KUKA KRL program: MyProgram_250().src

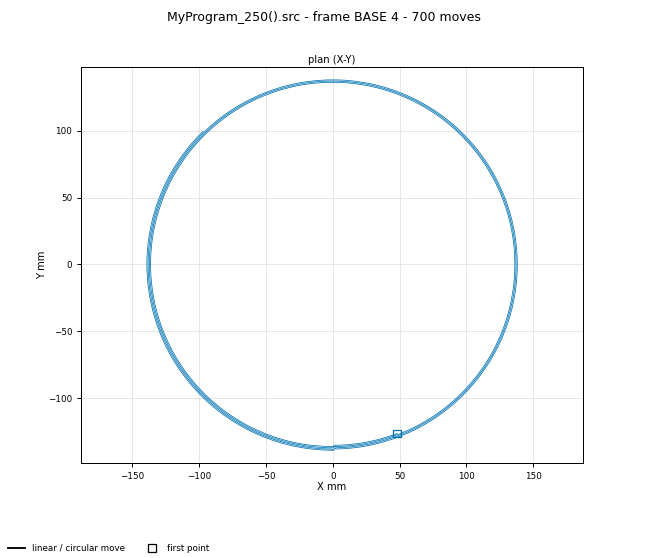
[picture p0: tool path of MyProgram_250().src in frame BASE 4, 700 of 700 moves have a stored position in this frame; points joined in program order, loops and branches not executed]
&ACCESS RVP
&REL 1
&PARAM TEMPLATE = C:\KRC\Roboter\Template\vorgabe
&PARAM EDITMASK = *
DEF MyProgram_250()
; ---- Setting reference (Base) ----
$BASE = BASE_DATA[4]

; --------------------------
; ---- Setting tool (TCP) ----
$TOOL = TOOL_DATA[3]
; --------------------------

$VEL.CP = VEL_APROX_PRINT
Startdeposition()
$VEL.CP = VEL_PRINT
LIN {X 48.2908,Y -126.5409,Z 164,A -68.332,B 12.277,C 0.2412,E1 12.3361,E2 518.7621} C_DIS
LIN {X 45.6625,Y -127.5105,Z 164,A -69.5545,B 12.2769,C 0.2436,E1 12.3329,E2 519.99} C_DIS
LIN {X 42.0708,Y -128.7422,Z 164,A -71.1085,B 12.2769,C 0.2439,E1 12.3288,E2 521.5389} C_DIS
LIN {X 38.9153,Y -129.7308,Z 164,A -72.4885,B 12.2769,C 0.2447,E1 12.3251,E2 522.9177} C_DIS
LIN {X 35.7562,Y -130.6369,Z 164,A -73.8812,B 12.2769,C 0.2461,E1 12.3214,E2 524.3117} C_DIS
LIN {X 32.9488,Y -131.3715,Z 164,A -75.1311,B 12.2769,C 0.2478,E1 12.318,E2 525.5653} C_DIS
LIN {X 29.371,Y -132.2193,Z 164,A -76.6506,B 12.2768,C 0.248,E1 12.3139,E2 527.0815} C_DIS
LIN {X 26.2188,Y -132.8803,Z 164,A -78.0066,B 12.2768,C 0.2489,E1 12.3102,E2 528.4377} C_DIS
LIN {X 23.2474,Y -133.4313,Z 164,A -79.2594,B 12.2768,C 0.249,E1 12.3067,E2 529.688} C_DIS
LIN {X 19.9409,Y -133.9663,Z 164,A -80.6907,B 12.2768,C 0.2502,E1 12.3028,E2 531.1221} C_DIS
LIN {X 16.8205,Y -134.3937,Z 164,A -82.0176,B 12.2768,C 0.2508,E1 12.2991,E2 532.4492} C_DIS
LIN {X 13.7158,Y -134.746,Z 164,A -83.3348,B 12.2768,C 0.2513,E1 12.2954,E2 533.7665} C_DIS
LIN {X 10.87,Y -135.0042,Z 164,A -84.525,B 12.2768,C 0.2513,E1 12.2921,E2 534.9551} C_DIS
LIN {X 7.9689,Y -135.2059,Z 164,A -85.7974,B 12.2768,C 0.2528,E1 12.2886,E2 536.2334} C_DIS
LIN {X 4.5191,Y -135.3668,Z 164,A -87.2223,B 12.2768,C 0.2522,E1 12.2846,E2 537.6546} C_DIS
LIN {X 0.9829,Y -135.4364,Z 164,A -88.496,B 12.2768,C 0.2465,E1 12.2811,E2 538.9014} C_DIS
Enddeposition()
LIN {X 0.9829,Y -135.4364,Z 164,A -88.496,B 12.2768,C 0.2465,E1 12.2811,E2 538.9014} C_DIS
Startdeposition()
$VEL.CP = VEL_PRINT
LIN {X 1.1754,Y -136.3554,Z 164,A -87.5778,B 12.2004,C 0.236,E1 12.2073,E2 537.9358} C_DIS
LIN {X 5.011,Y -136.268,Z 164,A -86.5742,B 12.2001,C 0.252,E1 12.2098,E2 537.0086} C_DIS
LIN {X 9.3611,Y -136.0392,Z 164,A -84.1098,B 12.2004,C 0.2343,E1 12.2169,E2 534.4629} C_DIS
LIN {X 13.3056,Y -135.7092,Z 164,A -82.8957,B 12.2002,C 0.2458,E1 12.2201,E2 533.3049} C_DIS
LIN {X 17.0554,Y -135.2905,Z 164,A -81.1665,B 12.2002,C 0.2411,E1 12.2249,E2 531.5566} C_DIS
LIN {X 20.8387,Y -134.7579,Z 164,A -79.6734,B 12.2002,C 0.2433,E1 12.229,E2 530.0767} C_DIS
LIN {X 24.8084,Y -134.0861,Z 164,A -77.9252,B 12.2003,C 0.2406,E1 12.2338,E2 528.3202} C_DIS
LIN {X 27.9166,Y -133.4733,Z 164,A -76.7034,B 12.2003,C 0.2427,E1 12.2372,E2 527.1114} C_DIS
LIN {X 30.4077,Y -132.9258,Z 164,A -75.5929,B 12.2003,C 0.2407,E1 12.2402,E2 525.9951} C_DIS
LIN {X 33.7097,Y -132.1272,Z 164,A -74.1914,B 12.2003,C 0.2402,E1 12.244,E2 524.5958} C_DIS
LIN {X 36.6449,Y -131.3432,Z 164,A -72.8971,B 12.2003,C 0.2386,E1 12.2475,E2 523.2983} C_DIS
LIN {X 40.6848,Y -130.1509,Z 164,A -71.1725,B 12.2003,C 0.2381,E1 12.2521,E2 521.5782} C_DIS
LIN {X 43.4948,Y -129.2373,Z 164,A -69.9381,B 12.2003,C 0.237,E1 12.2554,E2 520.3436} C_DIS
LIN {X 46.722,Y -128.1061,Z 164,A -68.506,B 12.2004,C 0.2355,E1 12.2591,E2 518.9109} C_DIS
LIN {X 49.6795,Y -126.9878,Z 164,A -67.1784,B 12.2004,C 0.2339,E1 12.2626,E2 517.5824} C_DIS
LIN {X 53.377,Y -125.4806,Z 164,A -65.5189,B 12.2004,C 0.2323,E1 12.2669,E2 515.9237} C_DIS
LIN {X 56.1528,Y -124.2617,Z 164,A -64.2407,B 12.2005,C 0.2305,E1 12.2701,E2 514.6438} C_DIS
LIN {X 60.2052,Y -122.3486,Z 164,A -62.1678,B 12.2006,C 0.2225,E1 12.2754,E2 512.5451} C_DIS
LIN {X 64.1876,Y -120.31,Z 164,A -60.4796,B 12.2006,C 0.2251,E1 12.2795,E2 510.8796} C_DIS
LIN {X 67.2225,Y -118.6409,Z 164,A -58.9313,B 12.2006,C 0.2202,E1 12.2833,E2 509.318} C_DIS
LIN {X 71.1825,Y -116.3076,Z 164,A -57.0303,B 12.2007,C 0.2179,E1 12.2879,E2 507.419} C_DIS
LIN {X 76.8995,Y -112.6097,Z 164,A -54.2881,B 12.2007,C 0.2164,E1 12.2943,E2 504.689} C_DIS
LIN {X 80.1373,Y -110.3286,Z 164,A -52.5882,B 12.2008,C 0.2123,E1 12.2981,E2 502.9829} C_DIS
LIN {X 83.4574,Y -107.839,Z 164,A -50.8412,B 12.2008,C 0.2089,E1 12.302,E2 501.2336} C_DIS
LIN {X 86.7001,Y -105.2501,Z 164,A -49.0457,B 12.201,C 0.2039,E1 12.3059,E2 499.4297} C_DIS
LIN {X 90.2463,Y -102.2252,Z 164,A -47.1321,B 12.201,C 0.2012,E1 12.3099,E2 497.5197} C_DIS
LIN {X 93.5477,Y -99.2129,Z 164,A -45.3151,B 12.201,C 0.199,E1 12.3136,E2 495.7083} C_DIS
LIN {X 96.533,Y -96.3111,Z 164,A -43.5592,B 12.2011,C 0.1951,E1 12.3171,E2 493.9497} C_DIS
LIN {X 99.5558,Y -93.1834,Z 164,A -41.2789,B 12.2014,C 0.1777,E1 12.3216,E2 491.6097} C_DIS
LIN {X 102.6887,Y -89.7185,Z 164,A -39.8828,B 12.2012,C 0.1898,E1 12.3241,E2 490.2835} C_DIS
LIN {X 106.8768,Y -84.6866,Z 164,A -37.2703,B 12.2012,C 0.1873,E1 12.3287,E2 487.6854} C_DIS
LIN {X 110.0508,Y -80.5187,Z 164,A -34.9862,B 12.2013,C 0.1796,E1 12.3326,E2 485.3884} C_DIS
LIN {X 112.1141,Y -77.6202,Z 164,A -33.4583,B 12.2014,C 0.1749,E1 12.335,E2 483.8546} C_DIS
LIN {X 114.4786,Y -74.0883,Z 164,A -31.6477,B 12.2014,C 0.1696,E1 12.3378,E2 482.0387} C_DIS
LIN {X 116.7798,Y -70.4053,Z 164,A -29.8574,B 12.2015,C 0.1659,E1 12.3404,E2 480.2506} C_DIS
LIN {X 118.8236,Y -66.898,Z 164,A -28.1541,B 12.2015,C 0.1615,E1 12.3428,E2 478.5456} C_DIS
LIN {X 121.0055,Y -62.8639,Z 164,A -26.1017,B 12.2017,C 0.1526,E1 12.3455,E2 476.4749} C_DIS
LIN {X 123.7331,Y -57.3059,Z 164,A -23.6996,B 12.2017,C 0.1514,E1 12.3483,E2 474.0949} C_DIS
LIN {X 125.3016,Y -53.7911,Z 164,A -22.153,B 12.2017,C 0.149,E1 12.3501,E2 472.5554} C_DIS
LIN {X 126.9426,Y -49.7956,Z 164,A -20.1796,B 12.2019,C 0.1393,E1 12.3521,E2 470.5597} C_DIS
LIN {X 128.4672,Y -45.7204,Z 164,A -18.565,B 12.2019,C 0.1405,E1 12.3536,E2 468.9701} C_DIS
LIN {X 129.6221,Y -42.339,Z 164,A -16.9303,B 12.2019,C 0.1322,E1 12.3551,E2 467.3168} C_DIS
LIN {X 130.8644,Y -38.3198,Z 164,A -15.3357,B 12.2019,C 0.1322,E1 12.3564,E2 465.7418} C_DIS
LIN {X 131.7544,Y -35.138,Z 164,A -13.9371,B 12.2019,C 0.128,E1 12.3574,E2 464.3403} C_DIS
LIN {X 132.7794,Y -31.0487,Z 164,A -12.2707,B 12.202,C 0.1259,E1 12.3585,E2 462.6851} C_DIS
LIN {X 133.6162,Y -27.2146,Z 164,A -10.3755,B 12.2021,C 0.1138,E1 12.3596,E2 460.7568} C_DIS
LIN {X 134.5659,Y -22.0482,Z 164,A -8.5679,B 12.2021,C 0.1192,E1 12.3605,E2 458.9971} C_DIS
LIN {X 134.9692,Y -19.4238,Z 164,A -7.2771,B 12.2021,C 0.1107,E1 12.361,E2 457.6829} C_DIS
LIN {X 135.4378,Y -15.8324,Z 164,A -5.6973,B 12.2022,C 0.1045,E1 12.3615,E2 456.0941} C_DIS
LIN {X 135.9509,Y -10.5712,Z 164,A -3.3772,B 12.2022,C 0.095,E1 12.3621,E2 453.7591} C_DIS
LIN {X 136.2584,Y -5.2565,Z 164,A -1.3986,B 12.2022,C 0.096,E1 12.3624,E2 451.8104} C_DIS
LIN {X 136.3511,Y -1.6569,Z 164,A 0.6013,B 12.2024,C 0.077,E1 12.3624,E2 449.7474} C_DIS
LIN {X 136.3329,Y 2.7517,Z 164,A 2.035,B 12.2024,C 0.084,E1 12.3624,E2 448.3646} C_DIS
LIN {X 136.0966,Y 8.4677,Z 164,A 4.3122,B 12.2024,C 0.0807,E1 12.3621,E2 446.1008} C_DIS
LIN {X 135.8407,Y 11.8936,Z 164,A 5.7832,B 12.2024,C 0.0756,E1 12.3617,E2 444.6249} C_DIS
LIN {X 135.3747,Y 16.3615,Z 164,A 7.552,B 12.2024,C 0.0736,E1 12.3612,E2 442.8689} C_DIS
LIN {X 134.8736,Y 20.0915,Z 164,A 9.3282,B 12.2024,C 0.0632,E1 12.3605,E2 441.0667} C_DIS
LIN {X 134.2268,Y 24.023,Z 164,A 10.8118,B 12.2024,C 0.064,E1 12.3598,E2 439.6054} C_DIS
LIN {X 133.6003,Y 27.2926,Z 164,A 12.2295,B 12.2025,C 0.0594,E1 12.359,E2 438.1839} C_DIS
LIN {X 132.8339,Y 30.8104,Z 164,A 13.82,B 12.2025,C 0.0528,E1 12.358,E2 436.5822} C_DIS
LIN {X 131.7281,Y 35.2364,Z 164,A 15.6314,B 12.2025,C 0.0504,E1 12.3568,E2 434.7822} C_DIS
LIN {X 130.7907,Y 38.5714,Z 164,A 17.007,B 12.2025,C 0.0487,E1 12.3557,E2 433.4153} C_DIS
LIN {X 129.6256,Y 42.3281,Z 164,A 18.626,B 12.2025,C 0.045,E1 12.3543,E2 431.7991} C_DIS
LIN {X 128.6051,Y 45.3331,Z 164,A 20.2475,B 12.2026,C 0.0329,E1 12.3528,E2 430.1404} C_DIS
LIN {X 126.6777,Y 50.467,Z 164,A 22.1375,B 12.2026,C 0.0387,E1 12.351,E2 428.3001} C_DIS
LIN {X 125.2088,Y 54.0057,Z 164,A 23.8065,B 12.2026,C 0.0326,E1 12.3492,E2 426.6224} C_DIS
LIN {X 123.8611,Y 57.029,Z 164,A 25.2775,B 12.2026,C 0.0266,E1 12.3474,E2 425.1403} C_DIS
LIN {X 122.1015,Y 60.7062,Z 164,A 26.9507,B 12.2026,C 0.0233,E1 12.3454,E2 423.4708} C_DIS
LIN {X 119.9975,Y 64.7693,Z 164,A 29.0703,B 12.2026,C 0.0126,E1 12.3426,E2 421.3252} C_DIS
LIN {X 117.4266,Y 69.3215,Z 164,A 31.0431,B 12.2026,C 0.0136,E1 12.3399,E2 419.3788} C_DIS
LIN {X 115.3058,Y 72.7938,Z 164,A 32.7303,B 12.2026,C 0.01,E1 12.3374,E2 417.6932} C_DIS
LIN {X 113.0619,Y 76.2328,Z 164,A 34.4602,B 12.2026,C 0.0057,E1 12.3347,E2 415.9616} C_DIS
LIN {X 110.1487,Y 80.3855,Z 164,A 36.5792,B 12.2026,C 0.001,E1 12.3313,E2 413.843} C_DIS
LIN {X 107.5201,Y 83.8688,Z 164,A 38.3945,B 12.2026,C -0.0027,E1 12.3282,E2 412.0288} C_DIS
LIN {X 104.8808,Y 87.1461,Z 164,A 40.1189,B 12.2026,C -0.0054,E1 12.3251,E2 410.3089} C_DIS
LIN {X 102.0458,Y 90.4492,Z 164,A 42.1318,B 12.2026,C -0.0147,E1 12.3214,E2 408.2722} C_DIS
LIN {X 99.2051,Y 93.556,Z 164,A 43.6393,B 12.2026,C -0.011,E1 12.3186,E2 406.7963} C_DIS
LIN {X 96.6273,Y 96.2162,Z 164,A 45.2671,B 12.2026,C -0.0162,E1 12.3154,E2 405.159} C_DIS
LIN {X 93.3106,Y 99.4366,Z 164,A 47.1839,B 12.2026,C -0.0193,E1 12.3115,E2 403.2445} C_DIS
LIN {X 90.041,Y 102.4067,Z 164,A 49.0558,B 12.2026,C -0.0233,E1 12.3076,E2 401.3699} C_DIS
LIN {X 82.6384,Y 108.4682,Z 164,A 52.8958,B 12.2026,C -0.0254,E1 12.2993,E2 397.5512} C_DIS
LIN {X 79.2735,Y 110.9509,Z 164,A 54.7025,B 12.2026,C -0.0298,E1 12.2952,E2 395.738} C_DIS
LIN {X 76.0068,Y 113.2143,Z 164,A 56.4444,B 12.2026,C -0.0345,E1 12.2912,E2 393.9867} C_DIS
LIN {X 72.4317,Y 115.5344,Z 164,A 58.2319,B 12.2026,C -0.0371,E1 12.287,E2 392.1994} C_DIS
LIN {X 68.7576,Y 117.7578,Z 164,A 60.021,B 12.2026,C -0.0393,E1 12.2827,E2 390.4118} C_DIS
LIN {X 64.8699,Y 119.9434,Z 164,A 61.8995,B 12.2026,C -0.042,E1 12.2781,E2 388.5325} C_DIS
LIN {X 60.8693,Y 122.021,Z 164,A 63.5625,B 12.2026,C -0.0381,E1 12.274,E2 386.8979} C_DIS
LIN {X 58.5741,Y 123.138,Z 164,A 64.7213,B 12.2026,C -0.0418,E1 12.2711,E2 385.7283} C_DIS
LIN {X 55.6269,Y 124.497,Z 164,A 66.0594,B 12.2026,C -0.0427,E1 12.2677,E2 384.3934} C_DIS
LIN {X 48.0521,Y 127.6123,Z 164,A 69.4891,B 12.2026,C -0.0459,E1 12.2588,E2 380.9654} C_DIS
LIN {X 43.7055,Y 129.1671,Z 164,A 71.365,B 12.2026,C -0.0459,E1 12.2539,E2 379.0976} C_DIS
LIN {X 40.232,Y 130.2896,Z 164,A 73.0275,B 12.2026,C -0.0507,E1 12.2494,E2 377.4195} C_DIS
LIN {X 36.7393,Y 131.3168,Z 164,A 74.5177,B 12.2026,C -0.0508,E1 12.2454,E2 375.9343} C_DIS
LIN {X 33.2881,Y 132.2341,Z 164,A 75.9811,B 12.2026,C -0.0508,E1 12.2415,E2 374.4757} C_DIS
LIN {X 29.6047,Y 133.1093,Z 164,A 77.5547,B 12.2026,C -0.0513,E1 12.2372,E2 372.9046} C_DIS
LIN {X 26.7382,Y 133.7131,Z 164,A 78.9283,B 12.2026,C -0.0558,E1 12.2334,E2 371.5138} C_DIS
LIN {X 20.8769,Y 134.752,Z 164,A 81.361,B 12.2026,C -0.055,E1 12.2267,E2 369.0902} C_DIS
LIN {X 17.6083,Y 135.218,Z 164,A 82.6906,B 12.2026,C -0.054,E1 12.2231,E2 367.7681} C_DIS
LIN {X 14.3853,Y 135.5989,Z 164,A 84.1121,B 12.2026,C -0.0559,E1 12.2191,E2 366.3399} C_DIS
LIN {X 9.93,Y 135.9977,Z 164,A 86.277,B 12.2025,C -0.0637,E1 12.213,E2 364.1407} C_DIS
LIN {X 6.2453,Y 136.218,Z 164,A 87.5863,B 12.2025,C -0.0575,E1 12.2094,E2 362.8618} C_DIS
LIN {X 2.09,Y 136.3439,Z 164,A 89.2131,B 12.2025,C -0.0544,E1 12.2049,E2 361.2504} C_DIS
LIN {X -2.8802,Y 136.3305,Z 164,A 91.4358,B 12.2025,C -0.0576,E1 12.1987,E2 359.0123} C_DIS
LIN {X -6.0127,Y 136.2289,Z 164,A 92.6748,B 12.2025,C -0.0554,E1 12.1952,E2 357.7837} C_DIS
LIN {X -9.8724,Y 136.0019,Z 164,A 94.2822,B 12.2025,C -0.0545,E1 12.1908,E2 356.1791} C_DIS
LIN {X -13.5412,Y 135.6866,Z 164,A 96.1288,B 12.2025,C -0.0617,E1 12.1855,E2 354.2968} C_DIS
LIN {X -17.0169,Y 135.2955,Z 164,A 97.2229,B 12.2025,C -0.0514,E1 12.1826,E2 353.2496} C_DIS
LIN {X -21.6342,Y 134.6347,Z 164,A 99.2182,B 12.2025,C -0.0514,E1 12.1771,E2 351.2512} C_DIS
LIN {X -25.9034,Y 133.8769,Z 164,A 101.1442,B 12.2025,C -0.0529,E1 12.1718,E2 349.3135} C_DIS
LIN {X -29.3192,Y 133.1713,Z 164,A 102.4765,B 12.2025,C -0.0485,E1 12.1682,E2 347.9986} C_DIS
LIN {X -31.9571,Y 132.5619,Z 164,A 103.6842,B 12.2025,C -0.0495,E1 12.1649,E2 346.7831} C_DIS
LIN {X -35.489,Y 131.6608,Z 164,A 105.1942,B 12.2025,C -0.0477,E1 12.1608,E2 345.2769} C_DIS
LIN {X -38.2408,Y 130.8875,Z 164,A 106.4065,B 12.2025,C -0.0469,E1 12.1576,E2 344.0641} C_DIS
LIN {X -41.5848,Y 129.8637,Z 164,A 108.3021,B 12.2025,C -0.0562,E1 12.1524,E2 342.1174} C_DIS
LIN {X -45.3778,Y 128.5896,Z 164,A 109.5797,B 12.2025,C -0.0443,E1 12.1491,E2 340.8907} C_DIS
LIN {X -48.6915,Y 127.3718,Z 164,A 111.2139,B 12.2025,C -0.0464,E1 12.1448,E2 339.2392} C_DIS
LIN {X -53.357,Y 125.4893,Z 164,A 113.1901,B 12.2025,C -0.0405,E1 12.1398,E2 337.2817} C_DIS
LIN {X -57.4791,Y 123.653,Z 164,A 115.1186,B 12.2025,C -0.0389,E1 12.1349,E2 335.3508} C_DIS
LIN {X -60.6509,Y 122.1288,Z 164,A 116.6044,B 12.2025,C -0.0371,E1 12.1311,E2 333.8655} C_DIS
LIN {X -64.1634,Y 120.3223,Z 164,A 118.1754,B 12.2026,C -0.0325,E1 12.1273,E2 332.3068} C_DIS
LIN {X -67.1054,Y 118.707,Z 164,A 119.7535,B 12.2026,C -0.0345,E1 12.1234,E2 330.7097} C_DIS
LIN {X -70.5956,Y 116.6647,Z 164,A 121.5191,B 12.2026,C -0.0335,E1 12.1191,E2 328.9376} C_DIS
LIN {X -75.2515,Y 113.7176,Z 164,A 123.5708,B 12.2026,C -0.0232,E1 12.1144,E2 326.9203} C_DIS
LIN {X -77.6775,Y 112.0743,Z 164,A 125.0837,B 12.2026,C -0.0279,E1 12.1108,E2 325.3742} C_DIS
LIN {X -81.3795,Y 109.4156,Z 164,A 127.1729,B 12.2026,C -0.0286,E1 12.1061,E2 323.2657} C_DIS
LIN {X -86.4616,Y 105.4458,Z 164,A 129.6546,B 12.2026,C -0.018,E1 12.1007,E2 320.8148} C_DIS
LIN {X -89.6471,Y 102.751,Z 164,A 131.4544,B 12.2026,C -0.0157,E1 12.0969,E2 319.0112} C_DIS
LIN {X -93.98,Y 98.804,Z 164,A 134.1578,B 12.2026,C -0.0163,E1 12.0913,E2 316.281} C_DIS
LIN {X -97.8786,Y 94.943,Z 164,A 136.2674,B 12.2026,C -0.0067,E1 12.0872,E2 314.1978} C_DIS
LIN {X -100.6527,Y 91.9976,Z 164,A 138.1624,B 12.2026,C -0.0075,E1 12.0836,E2 312.2809} C_DIS
LIN {X -103.5079,Y 88.7726,Z 164,A 139.7765,B 12.2026,C 0.0012,E1 12.0807,E2 310.6929} C_DIS
LIN {X -105.9909,Y 85.7926,Z 164,A 141.464,B 12.2026,C 0.0037,E1 12.0777,E2 309.0001} C_DIS
LIN {X -108.3883,Y 82.7427,Z 164,A 143.1293,B 12.2026,C 0.0067,E1 12.0748,E2 307.3324} C_DIS
LIN {X -110.9239,Y 79.3113,Z 164,A 144.9088,B 12.2026,C 0.0114,E1 12.0719,E2 305.5566} C_DIS
LIN {X -113.3119,Y 75.8606,Z 164,A 146.7387,B 12.2026,C 0.0143,E1 12.069,E2 303.7206} C_DIS
LIN {X -115.7364,Y 72.1074,Z 164,A 148.596,B 12.2026,C 0.0195,E1 12.0663,E2 301.868} C_DIS
LIN {X -117.8522,Y 68.5955,Z 164,A 150.3387,B 12.2026,C 0.0235,E1 12.0638,E2 300.1248} C_DIS
LIN {X -119.9202,Y 64.9131,Z 164,A 152.1972,B 12.2026,C 0.0262,E1 12.0613,E2 298.2582} C_DIS
LIN {X -121.7494,Y 61.4099,Z 164,A 153.7585,B 12.2026,C 0.0329,E1 12.0593,E2 296.711} C_DIS
LIN {X -123.1428,Y 58.5641,Z 164,A 155.0945,B 12.2026,C 0.0364,E1 12.0577,E2 295.376} C_DIS
LIN {X -124.7097,Y 55.1514,Z 164,A 156.6981,B 12.2026,C 0.0401,E1 12.0559,E2 293.7711} C_DIS
LIN {X -125.9443,Y 52.2683,Z 164,A 157.9973,B 12.2026,C 0.0442,E1 12.0544,E2 292.4757} C_DIS
LIN {X -127.3,Y 48.8763,Z 164,A 159.7004,B 12.2026,C 0.0446,E1 12.0527,E2 290.7538} C_DIS
LIN {X -130.2844,Y 40.2492,Z 164,A 163.2741,B 12.2025,C 0.0615,E1 12.0495,E2 287.217} C_DIS
LIN {X -131.6813,Y 35.4122,Z 164,A 165.3884,B 12.2025,C 0.0676,E1 12.0479,E2 285.1055} C_DIS
LIN {X -132.2734,Y 33.1333,Z 164,A 166.5437,B 12.2025,C 0.0667,E1 12.0471,E2 283.931} C_DIS
LIN {X -133.0087,Y 30.0448,Z 164,A 167.9427,B 12.2025,C 0.0691,E1 12.0462,E2 282.5256} C_DIS
LIN {X -133.7746,Y 26.4358,Z 164,A 169.6736,B 12.2025,C 0.0694,E1 12.0452,E2 280.7743} C_DIS
LIN {X -134.4969,Y 22.4613,Z 164,A 171.2578,B 12.2025,C 0.077,E1 12.0445,E2 279.2059} C_DIS
LIN {X -135.1097,Y 18.4347,Z 164,A 172.9444,B 12.2024,C 0.0826,E1 12.0438,E2 277.5244} C_DIS
LIN {X -135.5574,Y 14.7708,Z 164,A 174.654,B 12.2024,C 0.0835,E1 12.0433,E2 275.797} C_DIS
LIN {X -135.8857,Y 11.3605,Z 164,A 176.0931,B 12.2024,C 0.0878,E1 12.0429,E2 274.3596} C_DIS
LIN {X -136.1893,Y 6.8168,Z 164,A 177.9499,B 12.2023,C 0.0948,E1 12.0426,E2 272.5119} C_DIS
LIN {X -136.3248,Y 3.1531,Z 164,A 179.4669,B 12.2023,C 0.0999,E1 12.0425,E2 270.9995} C_DIS
LIN {X -136.3582,Y -0.6868,Z 164,A -178.8085,B 12.2023,C 0.1021,E1 12.0425,E2 269.2629} C_DIS
LIN {X -136.2686,Y -4.9965,Z 164,A -176.9851,B 12.2022,C 0.1072,E1 12.0426,E2 267.44} C_DIS
LIN {X -136.0777,Y -8.7749,Z 164,A -175.4217,B 12.2022,C 0.1124,E1 12.0429,E2 265.8816} C_DIS
LIN {X -135.7422,Y -12.9626,Z 164,A -173.6138,B 12.2021,C 0.1167,E1 12.0433,E2 264.0702} C_DIS
LIN {X -135.3736,Y -16.3707,Z 164,A -172.2277,B 12.2021,C 0.1221,E1 12.0437,E2 262.6923} C_DIS
LIN {X -134.944,Y -19.6,Z 164,A -170.768,B 12.2021,C 0.124,E1 12.0443,E2 261.2228} C_DIS
LIN {X -134.4164,Y -22.9437,Z 164,A -169.3405,B 12.202,C 0.128,E1 12.0449,E2 259.7961} C_DIS
LIN {X -133.6599,Y -26.9997,Z 164,A -167.5657,B 12.202,C 0.1321,E1 12.0459,E2 258.0179} C_DIS
LIN {X -132.8522,Y -30.73,Z 164,A -165.9037,B 12.202,C 0.1353,E1 12.0469,E2 256.3502} C_DIS
LIN {X -130.8835,Y -38.2546,Z 164,A -162.7074,B 12.2018,C 0.1463,E1 12.0492,E2 253.166} C_DIS
LIN {X -129.7971,Y -41.7935,Z 164,A -161.0607,B 12.2018,C 0.1485,E1 12.0506,E2 251.5094} C_DIS
LIN {X -128.1723,Y -46.5385,Z 164,A -158.8901,B 12.2018,C 0.1528,E1 12.0526,E2 249.3328} C_DIS
LIN {X -126.8925,Y -49.9245,Z 164,A -157.42,B 12.2016,C 0.1581,E1 12.0541,E2 247.8704} C_DIS
LIN {X -125.6054,Y -53.0798,Z 164,A -155.965,B 12.2016,C 0.1614,E1 12.0556,E2 246.4137} C_DIS
LIN {X -124.319,Y -56.0248,Z 164,A -154.1259,B 12.2016,C 0.1535,E1 12.0578,E2 244.5146} C_DIS
LIN {X -122.5111,Y -59.8758,Z 164,A -152.9286,B 12.2015,C 0.1721,E1 12.0592,E2 243.3924} C_DIS
LIN {X -121.5055,Y -61.8889,Z 164,A -151.8691,B 12.2015,C 0.1719,E1 12.0605,E2 242.3194} C_DIS
LIN {X -119.8259,Y -65.0861,Z 164,A -150.3428,B 12.2015,C 0.1756,E1 12.0625,E2 240.7932} C_DIS
LIN {X -117.9612,Y -68.4073,Z 164,A -148.5971,B 12.2014,C 0.1761,E1 12.065,E2 239.0307} C_DIS
LIN {X -115.6313,Y -72.2763,Z 164,A -146.666,B 12.2014,C 0.18,E1 12.0678,E2 237.0966} C_DIS
LIN {X -112.3824,Y -77.2308,Z 164,A -144.1988,B 12.2012,C 0.1865,E1 12.0716,E2 234.6339} C_DIS
LIN {X -109.8492,Y -80.7932,Z 164,A -142.2985,B 12.2012,C 0.1893,E1 12.0747,E2 232.7267} C_DIS
LIN {X -107.3054,Y -84.1424,Z 164,A -140.5351,B 12.2012,C 0.1934,E1 12.0778,E2 230.9649} C_DIS
LIN {X -104.5833,Y -87.5028,Z 164,A -138.593,B 12.2012,C 0.1944,E1 12.0812,E2 229.0081} C_DIS
LIN {X -102.3766,Y -90.075,Z 164,A -137.2836,B 12.201,C 0.2002,E1 12.0836,E2 227.7139} C_DIS
LIN {X -99.6679,Y -93.063,Z 164,A -135.57,B 12.201,C 0.2033,E1 12.0869,E2 225.9987} C_DIS
LIN {X -97.0183,Y -95.8227,Z 164,A -133.8879,B 12.201,C 0.2047,E1 12.0902,E2 224.3079} C_DIS
LIN {X -94.0628,Y -98.7249,Z 164,A -132.156,B 12.2009,C 0.2084,E1 12.0936,E2 222.5778} C_DIS
LIN {X -90.772,Y -101.759,Z 164,A -129.7114,B 12.2011,C 0.198,E1 12.0989,E2 220.0629} C_DIS
LIN {X -86.8596,Y -105.1181,Z 164,A -128.5277,B 12.2006,C 0.2261,E1 12.1011,E2 219.0035} C_DIS
LIN {X -83.2535,Y -107.997,Z 164,A -126.071,B 12.2007,C 0.2168,E1 12.1067,E2 216.4827} C_DIS
LIN {X -79.5121,Y -110.7802,Z 164,A -124.1355,B 12.2007,C 0.2206,E1 12.111,E2 214.5507} C_DIS
LIN {X -75.7632,Y -113.3769,Z 164,A -122.2299,B 12.2007,C 0.2238,E1 12.1154,E2 212.6468} C_DIS
LIN {X -72.1239,Y -115.7261,Z 164,A -120.4363,B 12.2006,C 0.2272,E1 12.1196,E2 210.8569} C_DIS
LIN {X -68.6534,Y -117.8187,Z 164,A -118.6976,B 12.2006,C 0.2287,E1 12.1238,E2 209.1139} C_DIS
LIN {X -64.8019,Y -119.9799,Z 164,A -116.7819,B 12.2006,C 0.2296,E1 12.1285,E2 207.1908} C_DIS
LIN {X -61.5596,Y -121.6732,Z 164,A -115.3776,B 12.2004,C 0.2348,E1 12.132,E2 205.8033} C_DIS
LIN {X -58.4721,Y -123.1867,Z 164,A -113.9328,B 12.2004,C 0.2365,E1 12.1356,E2 204.3586} C_DIS
LIN {X -50.3113,Y -126.7405,Z 164,A -110.2336,B 12.2003,C 0.2415,E1 12.1451,E2 200.6648} C_DIS
LIN {X -46.8174,Y -128.0717,Z 164,A -108.6754,B 12.2003,C 0.2433,E1 12.1492,E2 199.1082} C_DIS
LIN {X -43.4067,Y -129.2666,Z 164,A -106.9843,B 12.2003,C 0.2401,E1 12.1537,E2 197.3951} C_DIS
LIN {X -39.9183,Y -130.3856,Z 164,A -105.4121,B 12.2003,C 0.2404,E1 12.1579,E2 195.8186} C_DIS
LIN {X -34.7412,Y -131.8602,Z 164,A -103.248,B 12.2003,C 0.2444,E1 12.1637,E2 193.6665} C_DIS
LIN {X -31.5292,Y -132.665,Z 164,A -101.7848,B 12.2003,C 0.2433,E1 12.1677,E2 192.1939} C_DIS
LIN {X -27.3737,Y -133.5838,Z 164,A -99.6321,B 12.2004,C 0.2346,E1 12.1737,E2 189.9945} C_DIS
LIN {X -23.3491,Y -134.3473,Z 164,A -98.3049,B 12.2002,C 0.2457,E1 12.1772,E2 188.7169} C_DIS
LIN {X -19.2093,Y -134.9998,Z 164,A -96.5759,B 12.2002,C 0.247,E1 12.182,E2 186.9914} C_DIS
LIN {X -15.5778,Y -135.4681,Z 164,A -94.7869,B 12.2003,C 0.2408,E1 12.187,E2 185.1701} C_DIS
LIN {X -5.7775,Y -136.2381,Z 164,A -91.0439,B 12.2001,C 0.2514,E1 12.1973,E2 181.4747} C_DIS
LIN {X 0.9712,Y -136.3528,Z 164,A -89.3946,B 12.1994,C 0.2826,E1 12.2016,E2 179.9726} C_DIS
Enddeposition()
LIN {X 0.9712,Y -136.3528,Z 164,A -89.3948,B 12.1994,C 0.2826,E1 12.2016,E2 179.9728} C_DIS
Startdeposition()
$VEL.CP = VEL_PRINT
LIN {X 0.6652,Y -137.2779,Z 164,A -89.4096,B 12.1186,C 0.2916,E1 12.1208,E2 180.0344} C_DIS
LIN {X -4.5946,Y -137.2046,Z 164,A -91.0487,B 12.119,C 0.2772,E1 12.1164,E2 181.6049} C_DIS
LIN {X -7.9431,Y -137.0503,Z 164,A -92.7499,B 12.1188,C 0.285,E1 12.1115,E2 183.3447} C_DIS
LIN {X -11.6534,Y -136.7839,Z 164,A -93.9544,B 12.119,C 0.2758,E1 12.1083,E2 184.5061} C_DIS
LIN {X -17.3961,Y -136.1733,Z 164,A -96.3368,B 12.119,C 0.2746,E1 12.1017,E2 186.8858} C_DIS
LIN {X -20.6764,Y -135.7136,Z 164,A -98.8778,B 12.1183,C 0.304,E1 12.0943,E2 189.5716} C_DIS
LIN {X -28.5232,Y -134.284,Z 164,A -101.1177,B 12.119,C 0.2746,E1 12.0885,E2 191.6769} C_DIS
LIN {X -32.0412,Y -133.4876,Z 164,A -102.5474,B 12.119,C 0.2719,E1 12.0846,E2 193.0975} C_DIS
LIN {X -35.6795,Y -132.5618,Z 164,A -104.1585,B 12.119,C 0.272,E1 12.0803,E2 194.7145} C_DIS
LIN {X -39.8501,Y -131.3682,Z 164,A -105.965,B 12.1191,C 0.2707,E1 12.0754,E2 196.5207} C_DIS
LIN {X -43.2788,Y -130.2785,Z 164,A -107.4134,B 12.1191,C 0.2681,E1 12.0716,E2 197.9625} C_DIS
LIN {X -45.9692,Y -129.3551,Z 164,A -108.6792,B 12.1191,C 0.2691,E1 12.0682,E2 199.2385} C_DIS
LIN {X -49.2116,Y -128.1563,Z 164,A -110.1493,B 12.1191,C 0.2685,E1 12.0644,E2 200.712} C_DIS
LIN {X -52.7261,Y -126.7497,Z 164,A -112.0255,B 12.1191,C 0.2743,E1 12.0595,E2 202.6252} C_DIS
LIN {X -55.9951,Y -125.3397,Z 164,A -113.3309,B 12.1191,C 0.2682,E1 12.0562,E2 203.9082} C_DIS
LIN {X -60.4052,Y -123.2754,Z 164,A -115.2051,B 12.1193,C 0.2619,E1 12.0515,E2 205.7625} C_DIS
LIN {X -63.4248,Y -121.7496,Z 164,A -116.6706,B 12.1193,C 0.2615,E1 12.0478,E2 207.2346} C_DIS
LIN {X -67.1615,Y -119.7305,Z 164,A -118.4996,B 12.1193,C 0.2606,E1 12.0434,E2 209.0705} C_DIS
LIN {X -71.0553,Y -117.4614,Z 164,A -120.3772,B 12.1193,C 0.2579,E1 12.0388,E2 210.9474} C_DIS
LIN {X -74.7471,Y -115.1473,Z 164,A -122.2244,B 12.1194,C 0.2559,E1 12.0345,E2 212.7978} C_DIS
LIN {X -78.5407,Y -112.594,Z 164,A -124.1381,B 12.1194,C 0.2531,E1 12.0301,E2 214.7117} C_DIS
LIN {X -81.2834,Y -110.6302,Z 164,A -125.7437,B 12.1194,C 0.2556,E1 12.0264,E2 216.3417} C_DIS
LIN {X -84.7613,Y -107.9886,Z 164,A -127.3971,B 12.1196,C 0.2483,E1 12.0228,E2 217.9734} C_DIS
LIN {X -91.5082,Y -102.3342,Z 164,A -131.1075,B 12.1196,C 0.2426,E1 12.0149,E2 221.6872} C_DIS
LIN {X -94.7224,Y -99.3666,Z 164,A -132.958,B 12.1198,C 0.2396,E1 12.0111,E2 223.54} C_DIS
LIN {X -97.821,Y -96.3179,Z 164,A -134.7389,B 12.1198,C 0.2352,E1 12.0076,E2 225.316} C_DIS
LIN {X -100.6802,Y -93.3254,Z 164,A -136.5327,B 12.1198,C 0.2332,E1 12.0042,E2 227.1172} C_DIS
LIN {X -105.1397,Y -88.2705,Z 164,A -139.3383,B 12.12,C 0.227,E1 11.999,E2 229.9204} C_DIS
LIN {X -107.8167,Y -84.9802,Z 164,A -141.1311,B 12.12,C 0.2235,E1 11.9959,E2 231.715} C_DIS
LIN {X -111.3916,Y -80.2378,Z 164,A -144.5611,B 12.1197,C 0.24,E1 11.9901,E2 235.2606} C_DIS
LIN {X -115.3611,Y -74.4177,Z 164,A -146.6514,B 12.1202,C 0.2132,E1 11.987,E2 237.2446} C_DIS
LIN {X -117.7598,Y -70.5604,Z 164,A -148.5657,B 12.1203,C 0.209,E1 11.9842,E2 239.1599} C_DIS
LIN {X -119.7834,Y -67.0674,Z 164,A -150.1855,B 12.1204,C 0.2032,E1 11.982,E2 240.7705} C_DIS
LIN {X -121.8192,Y -63.2923,Z 164,A -152.0421,B 12.1204,C 0.2002,E1 11.9796,E2 242.6339} C_DIS
LIN {X -123.551,Y -59.843,Z 164,A -153.7912,B 12.1204,C 0.1992,E1 11.9774,E2 244.3989} C_DIS
LIN {X -125.7032,Y -55.1795,Z 164,A -155.8716,B 12.1206,C 0.1921,E1 11.975,E2 246.4698} C_DIS
LIN {X -127.1126,Y -51.8481,Z 164,A -157.3418,B 12.1206,C 0.1871,E1 11.9735,E2 247.9339} C_DIS
LIN {X -128.3163,Y -48.7945,Z 164,A -158.6047,B 12.1208,C 0.1809,E1 11.9722,E2 249.1824} C_DIS
LIN {X -130.3405,Y -43.0926,Z 164,A -161.8138,B 12.1206,C 0.1896,E1 11.9692,E2 252.4733} C_DIS
LIN {X -131.7763,Y -38.4779,Z 164,A -163.8591,B 12.1207,C 0.1846,E1 11.9676,E2 254.5202} C_DIS
LIN {X -133.0575,Y -33.7825,Z 164,A -165.2919,B 12.121,C 0.1652,E1 11.9667,E2 255.8777} C_DIS
LIN {X -133.9082,Y -30.237,Z 164,A -166.8824,B 12.121,C 0.1624,E1 11.9656,E2 257.4752} C_DIS
LIN {X -134.7991,Y -25.9772,Z 164,A -168.6796,B 12.121,C 0.1567,E1 11.9646,E2 259.2683} C_DIS
LIN {X -135.3706,Y -22.8129,Z 164,A -170.0782,B 12.1211,C 0.1541,E1 11.964,E2 260.6725} C_DIS
LIN {X -135.8325,Y -19.8835,Z 164,A -171.2435,B 12.1211,C 0.1489,E1 11.9635,E2 261.8277} C_DIS
LIN {X -136.297,Y -16.3931,Z 164,A -172.816,B 12.1212,C 0.147,E1 11.9629,E2 263.4113} C_DIS
LIN {X -136.712,Y -12.484,Z 164,A -174.5383,B 12.1212,C 0.144,E1 11.9625,E2 265.142} C_DIS
LIN {X -137.0214,Y -8.4123,Z 164,A -176.2132,B 12.1213,C 0.1383,E1 11.9621,E2 266.8115} C_DIS
LIN {X -137.2163,Y -4.1793,Z 164,A -178.0357,B 12.1213,C 0.1343,E1 11.9619,E2 268.6387} C_DIS
LIN {X -137.2692,Y 1.7564,Z 164,A 179.4607,B 12.1214,C 0.1276,E1 11.9619,E2 271.1428} C_DIS
LIN {X -137.17,Y 5.4819,Z 164,A 177.9158,B 12.1214,C 0.1228,E1 11.9621,E2 272.6846} C_DIS
LIN {X -136.9789,Y 9.1011,Z 164,A 176.3741,B 12.1215,C 0.119,E1 11.9623,E2 274.2283} C_DIS
LIN {X -136.4838,Y 14.7574,Z 164,A 173.9813,B 12.1215,C 0.1125,E1 11.9629,E2 276.6212} C_DIS
LIN {X -135.9839,Y 18.8239,Z 164,A 172.231,B 12.1216,C 0.1084,E1 11.9636,E2 278.3745} C_DIS
LIN {X -135.5193,Y 21.9215,Z 164,A 170.8991,B 12.1216,C 0.1051,E1 11.9641,E2 279.708} C_DIS
LIN {X -134.961,Y 25.1302,Z 164,A 169.4566,B 12.1216,C 0.103,E1 11.9649,E2 281.1591} C_DIS
LIN {X -134.1821,Y 28.9955,Z 164,A 167.9712,B 12.1217,C 0.0946,E1 11.9657,E2 282.6229} C_DIS
LIN {X -133.4458,Y 32.2145,Z 164,A 166.4753,B 12.1217,C 0.0932,E1 11.9667,E2 284.1316} C_DIS
LIN {X -132.3431,Y 36.4841,Z 164,A 164.541,B 12.1217,C 0.0901,E1 11.9681,E2 286.0752} C_DIS
LIN {X -131.0925,Y 40.751,Z 164,A 162.702,B 12.1217,C 0.0844,E1 11.9695,E2 287.91} C_DIS
LIN {X -129.015,Y 46.9124,Z 164,A 160.1499,B 12.1219,C 0.0731,E1 11.9718,E2 290.4392} C_DIS
LIN {X -127.2944,Y 51.3969,Z 164,A 158.0639,B 12.1219,C 0.0693,E1 11.974,E2 292.5328} C_DIS
LIN {X -125.8963,Y 54.733,Z 164,A 156.4546,B 12.1219,C 0.0674,E1 11.9757,E2 294.1525} C_DIS
LIN {X -124.3104,Y 58.2486,Z 164,A 154.8364,B 12.1219,C 0.0633,E1 11.9776,E2 295.7699} C_DIS
LIN {X -122.5467,Y 61.8708,Z 164,A 153.111,B 12.1219,C 0.0598,E1 11.9797,E2 297.4986} C_DIS
LIN {X -120.7164,Y 65.374,Z 164,A 151.3556,B 12.1219,C 0.0578,E1 11.9821,E2 299.2651} C_DIS
LIN {X -118.524,Y 69.269,Z 164,A 149.4681,B 12.1219,C 0.0535,E1 11.9847,E2 301.153} C_DIS
LIN {X -116.1689,Y 73.1494,Z 164,A 147.5626,B 12.1219,C 0.0489,E1 11.9875,E2 303.0577} C_DIS
LIN {X -113.5755,Y 77.1147,Z 164,A 145.6306,B 12.122,C 0.0429,E1 11.9904,E2 304.9818} C_DIS
LIN {X -111.4411,Y 80.169,Z 164,A 143.9527,B 12.122,C 0.0419,E1 11.9932,E2 306.6728} C_DIS
LIN {X -108.7689,Y 83.7588,Z 164,A 142.0961,B 12.122,C 0.0371,E1 11.9963,E2 308.526} C_DIS
LIN {X -105.9975,Y 87.2395,Z 164,A 140.0701,B 12.122,C 0.0367,E1 11.9999,E2 310.5703} C_DIS
LIN {X -100.7539,Y 93.2462,Z 164,A 136.9079,B 12.122,C 0.0254,E1 12.0057,E2 313.7087} C_DIS
LIN {X -95.9492,Y 98.1827,Z 164,A 134.2582,B 12.122,C 0.0139,E1 12.0109,E2 316.3279} C_DIS
LIN {X -91.029,Y 102.7608,Z 164,A 130.9454,B 12.122,C 0.0201,E1 12.0178,E2 319.6994} C_DIS
LIN {X -88.5386,Y 104.9142,Z 164,A 129.536,B 12.122,C 0.0182,E1 12.0208,E2 321.1116} C_DIS
LIN {X -85.8769,Y 107.1043,Z 164,A 127.6276,B 12.122,C 0.0265,E1 12.0251,E2 323.0751} C_DIS
LIN {X -81.2553,Y 110.6508,Z 164,A 125.8623,B 12.122,C 0.0064,E1 12.0289,E2 324.7577} C_DIS
LIN {X -78.8345,Y 112.389,Z 164,A 123.9335,B 12.122,C 0.0204,E1 12.0335,E2 326.7678} C_DIS
LIN {X -74.0323,Y 115.6082,Z 164,A 121.9152,B 12.122,C 0.0071,E1 12.0381,E2 328.7364} C_DIS
LIN {X -70.9672,Y 117.5147,Z 164,A 120.6785,B 12.122,C -0.0018,E1 12.041,E2 329.939} C_DIS
LIN {X -67.331,Y 119.6352,Z 164,A 118.8797,B 12.122,C -0.0034,E1 12.0453,E2 331.7412} C_DIS
LIN {X -63.8011,Y 121.552,Z 164,A 116.9513,B 12.122,C 0.0002,E1 12.0502,E2 333.6985} C_DIS
LIN {X -60.6179,Y 123.1705,Z 164,A 115.8834,B 12.122,C -0.0121,E1 12.0527,E2 334.7138} C_DIS
LIN {X -57.8699,Y 124.4855,Z 164,A 114.5168,B 12.122,C -0.0114,E1 12.0562,E2 336.0908} C_DIS
LIN {X -54.7385,Y 125.8939,Z 164,A 113.2944,B 12.122,C -0.0184,E1 12.0592,E2 337.2864} C_DIS
LIN {X -48.6841,Y 128.3577,Z 164,A 109.1831,B 12.122,C 0.0121,E1 12.0704,E2 341.5621} C_DIS
LIN {X -41.2346,Y 130.941,Z 164,A 106.9578,B 12.122,C -0.017,E1 12.0759,E2 343.6569} C_DIS
LIN {X -37.2946,Y 132.1165,Z 164,A 105.3301,B 12.122,C -0.0208,E1 12.0802,E2 345.2726} C_DIS
LIN {X -34.0269,Y 132.9955,Z 164,A 104.0178,B 12.122,C -0.0244,E1 12.0837,E2 346.5717} C_DIS
LIN {X -31.0944,Y 133.7123,Z 164,A 102.5467,B 12.122,C -0.0201,E1 12.0878,E2 348.0676} C_DIS
LIN {X -27.4999,Y 134.4966,Z 164,A 101.1055,B 12.122,C -0.0235,E1 12.0917,E2 349.4963} C_DIS
LIN {X -24.408,Y 135.0921,Z 164,A 99.7899,B 12.122,C -0.0242,E1 12.0953,E2 350.8112} C_DIS
LIN {X -21.4954,Y 135.5868,Z 164,A 98.5018,B 12.122,C -0.0235,E1 12.0989,E2 352.1053} C_DIS
LIN {X -18.7927,Y 135.9883,Z 164,A 96.5228,B 12.122,C -0.003,E1 12.1047,E2 354.1848} C_DIS
LIN {X -12.446,Y 136.7156,Z 164,A 94.5802,B 12.122,C -0.0221,E1 12.1098,E2 356.0388} C_DIS
LIN {X -8.4342,Y 137.02,Z 164,A 92.5867,B 12.122,C -0.0146,E1 12.1155,E2 358.0694} C_DIS
LIN {X -4.2413,Y 137.2146,Z 164,A 90.4756,B 12.122,C -0.0058,E1 12.1215,E2 360.2228} C_DIS
LIN {X 1.8351,Y 137.2679,Z 164,A 88.9017,B 12.122,C -0.0304,E1 12.1255,E2 361.6791} C_DIS
LIN {X 9.2309,Y 136.9707,Z 164,A 85.1446,B 12.122,C -0.0129,E1 12.1362,E2 365.5163} C_DIS
LIN {X 13.647,Y 136.6003,Z 164,A 83.7248,B 12.122,C -0.0236,E1 12.14,E2 366.8833} C_DIS
LIN {X 17.474,Y 136.1631,Z 164,A 82.3536,B 12.122,C -0.0293,E1 12.1438,E2 368.2251} C_DIS
LIN {X 24.9885,Y 134.9881,Z 164,A 78.8978,B 12.122,C -0.0206,E1 12.1534,E2 371.7146} C_DIS
LIN {X 28.3271,Y 134.3263,Z 164,A 77.551,B 12.122,C -0.0218,E1 12.157,E2 373.0519} C_DIS
LIN {X 31.7973,Y 133.5464,Z 164,A 76.0782,B 12.122,C -0.0212,E1 12.161,E2 374.523} C_DIS
LIN {X 35.4404,Y 132.6255,Z 164,A 74.6,B 12.122,C -0.0225,E1 12.165,E2 375.9898} C_DIS
LIN {X 38.2934,Y 131.8303,Z 164,A 73.3215,B 12.122,C -0.0205,E1 12.1684,E2 377.2734} C_DIS
LIN {X 41.5383,Y 130.844,Z 164,A 72.0402,B 12.122,C -0.0229,E1 12.1718,E2 378.5381} C_DIS
LIN {X 44.5089,Y 129.8642,Z 164,A 70.6301,B 12.122,C -0.0189,E1 12.1756,E2 379.9609} C_DIS
LIN {X 47.5757,Y 128.7728,Z 164,A 69.1577,B 12.122,C -0.0146,E1 12.1795,E2 381.4471} C_DIS
LIN {X 53.4064,Y 126.4655,Z 164,A 66.5594,B 12.122,C -0.0123,E1 12.1862,E2 384.043} C_DIS
LIN {X 57.3262,Y 124.7369,Z 164,A 64.8891,B 12.122,C -0.0135,E1 12.1904,E2 385.699} C_DIS
LIN {X 60.4024,Y 123.2768,Z 164,A 63.401,B 12.122,C -0.0099,E1 12.1942,E2 387.1953} C_DIS
LIN {X 63.4248,Y 121.7496,Z 164,A 62.0354,B 12.122,C -0.0094,E1 12.1976,E2 388.5552} C_DIS
LIN {X 67.199,Y 119.7094,Z 164,A 60.2158,B 12.122,C -0.0061,E1 12.202,E2 390.3786} C_DIS
LIN {X 71.1196,Y 117.4225,Z 164,A 58.3212,B 12.122,C -0.0034,E1 12.2066,E2 392.2735} C_DIS
LIN {X 75.019,Y 114.9708,Z 164,A 56.468,B 12.122,C -0.0023,E1 12.2109,E2 394.1186} C_DIS
LIN {X 78.5945,Y 112.5566,Z 164,A 54.579,B 12.122,C 0.003,E1 12.2153,E2 396.0189} C_DIS
LIN {X 82.4013,Y 109.8007,Z 164,A 52.6381,B 12.122,C 0.0058,E1 12.2196,E2 397.9578} C_DIS
LIN {X 87.3916,Y 105.8707,Z 164,A 49.9508,B 12.122,C 0.0116,E1 12.2255,E2 400.6503} C_DIS
LIN {X 91.1952,Y 102.6138,Z 164,A 47.9673,B 12.122,C 0.0126,E1 12.2297,E2 402.6216} C_DIS
LIN {X 93.9701,Y 100.0787,Z 164,A 46.2808,B 12.122,C 0.0189,E1 12.2331,E2 404.3231} C_DIS
LIN {X 97.6333,Y 96.5085,Z 164,A 44.3908,B 12.122,C 0.0164,E1 12.2368,E2 406.1839} C_DIS
LIN {X 102.6898,Y 91.1093,Z 164,A 41.2473,B 12.122,C 0.0245,E1 12.2428,E2 409.3359} C_DIS
LIN {X 105.5083,Y 87.8303,Z 164,A 39.4562,B 12.122,C 0.0282,E1 12.246,E2 411.1263} C_DIS
LIN {X 108.1385,Y 84.5705,Z 164,A 37.7362,B 12.122,C 0.0313,E1 12.249,E2 412.8438} C_DIS
LIN {X 110.8508,Y 80.9831,Z 164,A 35.8578,B 12.122,C 0.0357,E1 12.2522,E2 414.7235} C_DIS
LIN {X 113.6159,Y 77.055,Z 164,A 33.8582,B 12.122,C 0.0404,E1 12.2553,E2 416.7236} C_DIS
LIN {X 116.1173,Y 73.2311,Z 164,A 32.0339,B 12.122,C 0.0427,E1 12.2581,E2 418.5389} C_DIS
LIN {X 118.3094,Y 69.6342,Z 164,A 29.7638,B 12.122,C 0.0617,E1 12.2614,E2 420.8734} C_DIS
LIN {X 120.7047,Y 65.3955,Z 164,A 28.2079,B 12.122,C 0.0533,E1 12.2634,E2 422.3722} C_DIS
LIN {X 122.7267,Y 61.5173,Z 164,A 26.3522,B 12.122,C 0.0589,E1 12.2658,E2 424.233} C_DIS
LIN {X 124.5851,Y 57.6544,Z 164,A 24.7712,B 12.122,C 0.0576,E1 12.2676,E2 425.7895} C_DIS
LIN {X 125.736,Y 55.1036,Z 164,A 23.5676,B 12.122,C 0.0618,E1 12.269,E2 426.9985} C_DIS
LIN {X 127.3854,Y 51.1712,Z 164,A 21.2072,B 12.1218,C 0.0833,E1 12.2716,E2 429.432} C_DIS
LIN {X 129.2177,Y 46.3502,Z 164,A 19.714,B 12.1218,C 0.0702,E1 12.2729,E2 430.8457} C_DIS
LIN {X 130.3976,Y 42.9212,Z 164,A 18.1193,B 12.1218,C 0.0768,E1 12.2743,E2 432.4518} C_DIS
LIN {X 131.6528,Y 38.8996,Z 164,A 16.419,B 12.1218,C 0.08,E1 12.2757,E2 434.1465} C_DIS
LIN {X 132.6409,Y 35.3827,Z 164,A 14.8761,B 12.1218,C 0.0849,E1 12.2769,E2 435.6931} C_DIS
LIN {X 133.7781,Y 30.8066,Z 164,A 13.042,B 12.1218,C 0.0866,E1 12.2781,E2 437.5124} C_DIS
LIN {X 134.627,Y 26.859,Z 164,A 11.2361,B 12.1218,C 0.095,E1 12.2791,E2 439.335} C_DIS
LIN {X 135.3947,Y 22.6686,Z 164,A 9.6238,B 12.1218,C 0.0953,E1 12.2799,E2 440.9283} C_DIS
LIN {X 136.1576,Y 17.5158,Z 164,A 6.8513,B 12.1215,C 0.1191,E1 12.2809,E2 443.7774} C_DIS
LIN {X 136.7136,Y 12.4673,Z 164,A 5.3876,B 12.1216,C 0.1062,E1 12.2813,E2 445.1618} C_DIS
LIN {X 137.1101,Y 6.8151,Z 164,A 3.0039,B 12.1216,C 0.1137,E1 12.2817,E2 447.5504} C_DIS
LIN {X 137.2695,Y -1.7424,Z 164,A -0.5234,B 12.1215,C 0.123,E1 12.2819,E2 451.0761} C_DIS
LIN {X 136.9877,Y -8.9591,Z 164,A -4.2459,B 12.1211,C 0.1526,E1 12.2813,E2 454.89} C_DIS
LIN {X 136.4807,Y -14.7864,Z 164,A -5.8977,B 12.1213,C 0.1368,E1 12.2809,E2 456.4463} C_DIS
LIN {X 136.0425,Y -18.3945,Z 164,A -7.8648,B 12.1211,C 0.1544,E1 12.2801,E2 458.4714} C_DIS
LIN {X 135.4094,Y -22.5804,Z 164,A -9.7555,B 12.1211,C 0.1632,E1 12.2792,E2 460.3795} C_DIS
LIN {X 134.4748,Y -27.607,Z 164,A -11.2542,B 12.1211,C 0.1509,E1 12.2785,E2 461.8014} C_DIS
LIN {X 133.6366,Y -31.4231,Z 164,A -12.9438,B 12.1211,C 0.1574,E1 12.2774,E2 463.5004} C_DIS
LIN {X 132.7144,Y -35.1071,Z 164,A -14.4475,B 12.1211,C 0.1596,E1 12.2764,E2 464.9957} C_DIS
LIN {X 131.8924,Y -38.0814,Z 164,A -15.7511,B 12.121,C 0.1637,E1 12.2754,E2 466.3028} C_DIS
LIN {X 131.0187,Y -40.9913,Z 164,A -17.0154,B 12.121,C 0.1673,E1 12.2743,E2 467.5682} C_DIS
LIN {X 129.7121,Y -44.9475,Z 164,A -18.6247,B 12.121,C 0.1684,E1 12.2729,E2 469.1632} C_DIS
LIN {X 128.804,Y -47.4924,Z 164,A -20.5427,B 12.1205,C 0.1946,E1 12.271,E2 471.1815} C_DIS
LIN {X 126.6792,Y -52.895,Z 164,A -21.8614,B 12.1209,C 0.1692,E1 12.2697,E2 472.3646} C_DIS
LIN {X 124.3854,Y -58.0864,Z 164,A -24.1452,B 12.1209,C 0.1733,E1 12.2672,E2 474.6408} C_DIS
LIN {X 121.9077,Y -63.1239,Z 164,A -26.9545,B 12.1206,C 0.1933,E1 12.2636,E2 477.5119} C_DIS
LIN {X 119.7015,Y -67.2131,Z 164,A -28.8351,B 12.1206,C 0.1967,E1 12.261,E2 479.3875} C_DIS
LIN {X 117.2465,Y -71.4106,Z 164,A -30.8821,B 12.1204,C 0.2025,E1 12.2581,E2 481.439} C_DIS
LIN {X 114.8065,Y -75.27,Z 164,A -32.7441,B 12.1204,C 0.2061,E1 12.2553,E2 483.2978} C_DIS
LIN {X 112.8417,Y -78.1847,Z 164,A -34.1493,B 12.1204,C 0.208,E1 12.2531,E2 484.697} C_DIS
LIN {X 110.7604,Y -81.1056,Z 164,A -35.9987,B 12.1201,C 0.2219,E1 12.25,E2 486.5923} C_DIS
LIN {X 108.3082,Y -84.3532,Z 164,A -37.355,B 12.1201,C 0.2161,E1 12.2477,E2 487.9077} C_DIS
LIN {X 104.7903,Y -88.6855,Z 164,A -39.7085,B 12.1201,C 0.2223,E1 12.2435,E2 490.2669} C_DIS
LIN {X 101.7301,Y -92.1793,Z 164,A -41.5414,B 12.1201,C 0.2237,E1 12.2402,E2 492.0887} C_DIS
LIN {X 98.9574,Y -95.1506,Z 164,A -43.2366,B 12.12,C 0.2275,E1 12.2369,E2 493.7857} C_DIS
LIN {X 95.948,Y -98.1839,Z 164,A -44.9874,B 12.12,C 0.2305,E1 12.2334,E2 495.5344} C_DIS
LIN {X 92.9072,Y -101.0657,Z 164,A -46.7217,B 12.1199,C 0.2337,E1 12.2299,E2 497.2688} C_DIS
LIN {X 89.7218,Y -103.9041,Z 164,A -48.5033,B 12.1198,C 0.2374,E1 12.2262,E2 499.0524} C_DIS
LIN {X 86.3273,Y -106.7411,Z 164,A -50.324,B 12.1198,C 0.2403,E1 12.2222,E2 500.8718} C_DIS
LIN {X 83.0601,Y -109.3034,Z 164,A -52.0543,B 12.1197,C 0.2436,E1 12.2184,E2 502.6037} C_DIS
LIN {X 79.5085,Y -111.9134,Z 164,A -53.8887,B 12.1197,C 0.2468,E1 12.2142,E2 504.4393} C_DIS
LIN {X 75.8886,Y -114.3989,Z 164,A -55.5795,B 12.1197,C 0.2461,E1 12.2104,E2 506.114} C_DIS
LIN {X 69.4445,Y -118.4209,Z 164,A -58.8405,B 12.1195,C 0.2539,E1 12.2026,E2 509.3897} C_DIS
LIN {X 63.3154,Y -121.8071,Z 164,A -61.5175,B 12.1195,C 0.2515,E1 12.1961,E2 512.0384} C_DIS
LIN {X 58.0706,Y -124.3927,Z 164,A -64.1595,B 12.1193,C 0.2606,E1 12.1894,E2 514.7081} C_DIS
LIN {X 54.7754,Y -125.8779,Z 164,A -65.473,B 12.1193,C 0.2572,E1 12.1861,E2 515.9984} C_DIS
LIN {X 51.7114,Y -127.1676,Z 164,A -66.8948,B 12.1193,C 0.2599,E1 12.1824,E2 517.4257} C_DIS
LIN {X 49.0059,Y -128.2363,Z 164,A -68.3079,B 12.1192,C 0.2669,E1 12.1787,E2 518.865} C_DIS
LIN {X 45.6426,Y -129.4712,Z 164,A -69.7984,B 12.1192,C 0.2684,E1 12.1748,E2 520.3561} C_DIS
LIN {X 41.8894,Y -130.7319,Z 164,A -71.2855,B 12.1192,C 0.2656,E1 12.1709,E2 521.8236} C_DIS
LIN {X 39.1777,Y -131.5714,Z 164,A -72.4877,B 12.1192,C 0.2672,E1 12.1676,E2 523.029} C_DIS
LIN {X 35.6823,Y -132.561,Z 164,A -74.0114,B 12.1192,C 0.2688,E1 12.1635,E2 524.5547} C_DIS
LIN {X 32.6642,Y -133.3374,Z 164,A -75.3658,B 12.1191,C 0.2714,E1 12.1598,E2 525.9169} C_DIS
LIN {X 28.1069,Y -134.3731,Z 164,A -77.2121,B 12.1191,C 0.2701,E1 12.1548,E2 527.7514} C_DIS
LIN {X 23.5647,Y -135.243,Z 164,A -79.2626,B 12.1191,C 0.2747,E1 12.1492,E2 529.8184} C_DIS
LIN {X 20.1833,Y -135.7896,Z 164,A -80.6813,B 12.1191,C 0.2752,E1 12.1453,E2 531.2367} C_DIS
LIN {X 14.4975,Y -136.5118,Z 164,A -83.1958,B 12.1189,C 0.2796,E1 12.1382,E2 533.768} C_DIS
LIN {X 8.2363,Y -137.0322,Z 164,A -85.5357,B 12.1191,C 0.273,E1 12.1318,E2 536.0737} C_DIS
LIN {X 2.0442,Y -137.2644,Z 164,A -88.136,B 12.1191,C 0.274,E1 12.1246,E2 538.6773} C_DIS
LIN {X 2.0442,Y -137.2644,Z 164,A -88.136,B 12.1191,C 0.274,E1 12.1246,E2 538.6773} C_DIS
Enddeposition()
LIN {X 0.9857,Y -138.1868,Z 164,A -88.2522,B 11.8419,C 0.2873,E1 11.8472,E2 538.8703} C_DIS
Startdeposition()
$VEL.CP = VEL_PRINT
LIN {X 4.0366,Y -138.1402,Z 164,A -86.5305,B 11.8422,C 0.275,E1 11.8522,E2 537.0897} C_DIS
LIN {X 7.7902,Y -137.9811,Z 164,A -85.1177,B 11.8422,C 0.2785,E1 11.8561,E2 535.6947} C_DIS
LIN {X 13.9545,Y -137.494,Z 164,A -82.5556,B 11.8422,C 0.2776,E1 11.8633,E2 533.1314} C_DIS
LIN {X 18.528,Y -136.9525,Z 164,A -80.5101,B 11.8422,C 0.2729,E1 11.869,E2 531.0672} C_DIS
LIN {X 22.3622,Y -136.3782,Z 164,A -78.304,B 11.8426,C 0.2557,E1 11.8753,E2 528.7824} C_DIS
LIN {X 27.7381,Y -135.3866,Z 164,A -76.732,B 11.8422,C 0.273,E1 11.8793,E2 527.2991} C_DIS
LIN {X 31.1618,Y -134.6403,Z 164,A -75.1842,B 11.8423,C 0.2693,E1 11.8836,E2 525.738} C_DIS
LIN {X 35.0741,Y -133.675,Z 164,A -73.5475,B 11.8423,C 0.2688,E1 11.888,E2 524.1044} C_DIS
LIN {X 38.5604,Y -132.7104,Z 164,A -72.098,B 11.8423,C 0.2688,E1 11.8919,E2 522.6602} C_DIS
LIN {X 41.9568,Y -131.6758,Z 164,A -70.6512,B 11.8423,C 0.268,E1 11.8957,E2 521.2155} C_DIS
LIN {X 44.9727,Y -130.6768,Z 164,A -69.3418,B 11.8423,C 0.2668,E1 11.8992,E2 519.9061} C_DIS
LIN {X 47.9268,Y -129.6234,Z 164,A -67.9558,B 11.8425,C 0.2629,E1 11.9028,E2 518.508} C_DIS
LIN {X 51.5992,Y -128.2044,Z 164,A -66.5182,B 11.8424,C 0.2663,E1 11.9065,E2 517.0941} C_DIS
LIN {X 54.0479,Y -127.1943,Z 164,A -65.2657,B 11.8425,C 0.2607,E1 11.9098,E2 515.8209} C_DIS
LIN {X 57.6752,Y -125.5887,Z 164,A -63.8884,B 11.8425,C 0.2659,E1 11.9132,E2 514.4764} C_DIS
LIN {X 61.1092,Y -123.9536,Z 164,A -61.9748,B 11.8427,C 0.2543,E1 11.9181,E2 512.518} C_DIS
LIN {X 66.0376,Y -121.402,Z 164,A -59.7578,B 11.8427,C 0.2532,E1 11.9236,E2 510.3098} C_DIS
LIN {X 69.5178,Y -119.4435,Z 164,A -57.3864,B 11.8431,C 0.2303,E1 11.9296,E2 507.8438} C_DIS
LIN {X 74.8354,Y -116.186,Z 164,A -55.5422,B 11.8428,C 0.247,E1 11.9337,E2 506.0935} C_DIS
LIN {X 78.5654,Y -113.6972,Z 164,A -53.7155,B 11.8428,C 0.2446,E1 11.9379,E2 504.2691} C_DIS
LIN {X 82.1757,Y -111.1158,Z 164,A -51.8687,B 11.8429,C 0.241,E1 11.9421,E2 502.4195} C_DIS
LIN {X 85.5506,Y -108.5381,Z 164,A -50.1405,B 11.8429,C 0.2386,E1 11.9459,E2 500.6937} C_DIS
LIN {X 89.0398,Y -105.6947,Z 164,A -48.3461,B 11.843,C 0.2369,E1 11.9497,E2 498.9066} C_DIS
LIN {X 92.2163,Y -102.9346,Z 164,A -46.5942,B 11.843,C 0.2331,E1 11.9534,E2 497.1518} C_DIS
LIN {X 95.2425,Y -100.1417,Z 164,A -44.8725,B 11.8432,C 0.2291,E1 11.9569,E2 495.4265} C_DIS
LIN {X 98.3499,Y -97.092,Z 164,A -43.0515,B 11.8432,C 0.2247,E1 11.9605,E2 493.6014} C_DIS
LIN {X 101.7709,Y -93.4989,Z 164,A -40.778,B 11.8434,C 0.2139,E1 11.9649,E2 491.2976} C_DIS
LIN {X 104.1991,Y -90.785,Z 164,A -39.4354,B 11.8434,C 0.2152,E1 11.9673,E2 489.975} C_DIS
LIN {X 107.4517,Y -86.9111,Z 164,A -37.4855,B 11.8434,C 0.2145,E1 11.9708,E2 488.0417} C_DIS
LIN {X 109.5084,Y -84.3058,Z 164,A -35.6108,B 11.8437,C 0.1967,E1 11.9741,E2 486.1009} C_DIS
LIN {X 112.4223,Y -80.3778,Z 164,A -34.3124,B 11.8435,C 0.2129,E1 11.976,E2 484.8944} C_DIS
LIN {X 113.9063,Y -78.2606,Z 164,A -32.9911,B 11.8436,C 0.203,E1 11.9782,E2 483.5398} C_DIS
LIN {X 116.5697,Y -74.236,Z 164,A -31.1397,B 11.8436,C 0.2023,E1 11.981,E2 481.7053} C_DIS
LIN {X 118.2535,Y -71.5226,Z 164,A -29.7565,B 11.8437,C 0.1971,E1 11.983,E2 480.313} C_DIS
LIN {X 120.5857,Y -67.5168,Z 164,A -27.8429,B 11.8438,C 0.1923,E1 11.9856,E2 478.3981} C_DIS
LIN {X 122.7059,Y -63.5819,Z 164,A -25.817,B 11.844,C 0.1823,E1 11.9883,E2 476.3478} C_DIS
LIN {X 124.1457,Y -60.7198,Z 164,A -24.6784,B 11.844,C 0.1843,E1 11.9897,E2 475.232} C_DIS
LIN {X 126.051,Y -56.6572,Z 164,A -22.9842,B 11.844,C 0.184,E1 11.9916,E2 473.5569} C_DIS
LIN {X 127.3599,Y -53.6515,Z 164,A -21.6457,B 11.844,C 0.1809,E1 11.9931,E2 472.2196} C_DIS
LIN {X 129.743,Y -47.6048,Z 164,A -18.831,B 11.8441,C 0.1699,E1 11.996,E2 469.3864} C_DIS
LIN {X 131.0639,Y -43.831,Z 164,A -17.2837,B 11.8441,C 0.1684,E1 11.9973,E2 467.8511} C_DIS
LIN {X 132.0891,Y -40.6371,Z 164,A -15.9338,B 11.8442,C 0.1656,E1 11.9985,E2 466.5049} C_DIS
LIN {X 133.1318,Y -37.0787,Z 164,A -14.5499,B 11.8442,C 0.1656,E1 11.9995,E2 465.1389} C_DIS
LIN {X 133.9038,Y -34.1861,Z 164,A -13.1244,B 11.8443,C 0.1567,E1 12.0005,E2 463.6883} C_DIS
LIN {X 134.8907,Y -30.0652,Z 164,A -11.3374,B 11.8443,C 0.1507,E1 12.0017,E2 461.8955} C_DIS
LIN {X 135.8516,Y -25.3693,Z 164,A -9.1975,B 11.8445,C 0.1404,E1 12.0028,E2 459.7337} C_DIS
LIN {X 136.4401,Y -21.9909,Z 164,A -7.5215,B 11.8447,C 0.1287,E1 12.0036,E2 458.0233} C_DIS
LIN {X 137.1306,Y -17.169,Z 164,A -6.0638,B 11.8445,C 0.1394,E1 12.0041,E2 456.6356} C_DIS
LIN {X 137.8381,Y -9.9808,Z 164,A -2.826,B 11.8447,C 0.1234,E1 12.0049,E2 453.3633} C_DIS
LIN {X 138.0479,Y -6.4783,Z 164,A -1.5755,B 11.8447,C 0.1251,E1 12.005,E2 452.1374} C_DIS
LIN {X 138.1913,Y -1.6201,Z 164,A 0.2389,B 11.8447,C 0.1251,E1 12.0051,E2 450.3466} C_DIS
LIN {X 138.1464,Y 3.8144,Z 164,A 2.5302,B 11.8447,C 0.1172,E1 12.0051,E2 448.0479} C_DIS
LIN {X 137.7511,Y 11.1281,Z 164,A 5.4962,B 11.8448,C 0.1104,E1 12.0046,E2 445.0879} C_DIS
LIN {X 137.1838,Y 16.7233,Z 164,A 7.823,B 11.8448,C 0.1037,E1 12.0039,E2 442.7594} C_DIS
LIN {X 136.839,Y 19.3411,Z 164,A 9.2721,B 11.845,C 0.0901,E1 12.0033,E2 441.2639} C_DIS
LIN {X 136.2518,Y 23.1196,Z 164,A 10.5921,B 11.845,C 0.0933,E1 12.0027,E2 439.9762} C_DIS
LIN {X 135.5503,Y 26.9338,Z 164,A 11.9885,B 11.845,C 0.0949,E1 12.0019,E2 438.6053} C_DIS
LIN {X 134.82,Y 30.375,Z 164,A 13.5461,B 11.845,C 0.0878,E1 12.001,E2 437.0336} C_DIS
LIN {X 134.0119,Y 33.7603,Z 164,A 14.9587,B 11.845,C 0.0845,E1 12.0001,E2 435.6236} C_DIS
LIN {X 133.0838,Y 37.2501,Z 164,A 16.4018,B 11.845,C 0.0819,E1 11.999,E2 434.186} C_DIS
LIN {X 132.0268,Y 40.8409,Z 164,A 18.0011,B 11.8451,C 0.0762,E1 11.9977,E2 432.5792} C_DIS
LIN {X 130.663,Y 45.0124,Z 164,A 19.6489,B 11.8451,C 0.0761,E1 11.9963,E2 430.9517} C_DIS
LIN {X 129.8422,Y 47.3297,Z 164,A 20.993,B 11.8451,C 0.0639,E1 11.995,E2 429.5655} C_DIS
LIN {X 127.9936,Y 52.1223,Z 164,A 22.9558,B 11.8451,C 0.0629,E1 11.9929,E2 427.6222} C_DIS
LIN {X 126.2493,Y 56.214,Z 164,A 24.6593,B 11.8451,C 0.062,E1 11.9911,E2 425.9349} C_DIS
LIN {X 125.0185,Y 58.9045,Z 164,A 25.9874,B 11.8452,C 0.0559,E1 11.9895,E2 424.5932} C_DIS
LIN {X 123.3371,Y 62.3453,Z 164,A 27.476,B 11.8452,C 0.0546,E1 11.9876,E2 423.1159} C_DIS
LIN {X 121.5415,Y 65.7817,Z 164,A 29.2857,B 11.8452,C 0.0447,E1 11.9852,E2 421.2794} C_DIS
LIN {X 118.739,Y 70.7137,Z 164,A 31.4427,B 11.8452,C 0.0443,E1 11.9822,E2 419.1455} C_DIS
LIN {X 116.3762,Y 74.5382,Z 164,A 33.2497,B 11.8452,C 0.0414,E1 11.9795,E2 417.3445} C_DIS
LIN {X 114.0453,Y 78.0582,Z 164,A 35.0474,B 11.8452,C 0.0358,E1 11.9767,E2 415.5397} C_DIS
LIN {X 111.3129,Y 81.9074,Z 164,A 36.8899,B 11.8452,C 0.0345,E1 11.9737,E2 413.7105} C_DIS
LIN {X 108.9683,Y 85.0027,Z 164,A 38.5827,B 11.8453,C 0.0284,E1 11.9708,E2 412.0063} C_DIS
LIN {X 106.2425,Y 88.3856,Z 164,A 40.296,B 11.8453,C 0.0269,E1 11.9678,E2 410.3031} C_DIS
LIN {X 103.4303,Y 91.6601,Z 164,A 43.0162,B 11.8453,C -0.0034,E1 11.9626,E2 407.4637} C_DIS
LIN {X 98.54,Y 96.8982,Z 164,A 44.9885,B 11.8453,C 0.0187,E1 11.959,E2 405.6171} C_DIS
LIN {X 94.3518,Y 100.981,Z 164,A 47.47,B 11.8453,C 0.0123,E1 11.954,E2 403.1275} C_DIS
LIN {X 91.1529,Y 103.8782,Z 164,A 49.1458,B 11.8453,C 0.012,E1 11.9505,E2 401.4653} C_DIS
LIN {X 86.9207,Y 107.444,Z 164,A 51.4727,B 11.8453,C 0.0069,E1 11.9455,E2 399.1336} C_DIS
LIN {X 83.5612,Y 110.0774,Z 164,A 53.2922,B 11.8453,C 0.0024,E1 11.9414,E2 397.3074} C_DIS
LIN {X 79.8643,Y 112.788,Z 164,A 55.1857,B 11.8453,C -0.0005,E1 11.9372,E2 395.4143} C_DIS
LIN {X 76.0737,Y 115.3784,Z 164,A 57.059,B 11.8453,C -0.0027,E1 11.9328,E2 393.5444} C_DIS
LIN {X 72.1702,Y 117.8594,Z 164,A 58.9479,B 11.8453,C -0.0048,E1 11.9283,E2 391.6588} C_DIS
LIN {X 68.2511,Y 120.1717,Z 164,A 60.8352,B 11.8453,C -0.0076,E1 11.9238,E2 389.7711} C_DIS
LIN {X 64.6222,Y 122.1596,Z 164,A 62.4452,B 11.8453,C -0.007,E1 11.9199,E2 388.1741} C_DIS
LIN {X 61.3176,Y 123.8508,Z 164,A 64.0144,B 11.8453,C -0.0098,E1 11.9159,E2 386.601} C_DIS
LIN {X 58.5099,Y 125.2028,Z 164,A 65.3225,B 11.8453,C -0.0118,E1 11.9126,E2 385.2909} C_DIS
LIN {X 52.5689,Y 127.812,Z 164,A 67.9313,B 11.8453,C -0.0125,E1 11.906,E2 382.6924} C_DIS
LIN {X 49.3734,Y 129.0801,Z 164,A 69.369,B 11.8453,C -0.0143,E1 11.9022,E2 381.2532} C_DIS
LIN {X 45.4486,Y 130.5118,Z 164,A 71.1928,B 11.8453,C -0.0184,E1 11.8974,E2 379.418} C_DIS
LIN {X 40.9693,Y 131.9874,Z 164,A 73.0967,B 11.8453,C -0.0187,E1 11.8923,E2 377.5208} C_DIS
LIN {X 37.564,Y 132.9961,Z 164,A 74.537,B 11.8453,C -0.0189,E1 11.8885,E2 376.0846} C_DIS
LIN {X 34.0485,Y 133.9388,Z 164,A 76.0486,B 11.8453,C -0.0201,E1 11.8844,E2 374.573} C_DIS
LIN {X 29.8189,Y 134.9451,Z 164,A 77.887,B 11.8453,C -0.0221,E1 11.8794,E2 372.7306} C_DIS
LIN {X 26.4484,Y 135.6453,Z 164,A 79.3708,B 11.8453,C -0.0243,E1 11.8753,E2 371.24} C_DIS
LIN {X 19.2315,Y 136.8546,Z 164,A 82.4925,B 11.8453,C -0.0278,E1 11.8667,E2 368.1083} C_DIS
LIN {X 15.1205,Y 137.3697,Z 164,A 84.1257,B 11.8453,C -0.0261,E1 11.8622,E2 366.4862} C_DIS
LIN {X 9.6554,Y 137.8619,Z 164,A 86.1862,B 11.8453,C -0.0209,E1 11.8565,E2 364.4534} C_DIS
LIN {X 5.8962,Y 138.0742,Z 164,A 87.8673,B 11.8453,C -0.0242,E1 11.8518,E2 362.758} C_DIS
LIN {X 1.3188,Y 138.1939,Z 164,A 90.3021,B 11.8453,C -0.0379,E1 11.8448,E2 360.257} C_DIS
LIN {X -3.613,Y 138.152,Z 164,A 91.7128,B 11.8453,C -0.0214,E1 11.8411,E2 358.9265} C_DIS
LIN {X -11.3549,Y 137.732,Z 164,A 94.7494,B 11.8453,C -0.0161,E1 11.8327,E2 355.9138} C_DIS
LIN {X -18.7809,Y 136.919,Z 164,A 98.234,B 11.8453,C -0.0246,E1 11.8229,E2 352.3833} C_DIS
LIN {X -23.4471,Y 136.1971,Z 164,A 100.069,B 11.8453,C -0.0205,E1 11.8179,E2 350.5648} C_DIS
LIN {X -27.4146,Y 135.4525,Z 164,A 101.6914,B 11.8453,C -0.0182,E1 11.8134,E2 348.9497} C_DIS
LIN {X -30.8268,Y 134.7168,Z 164,A 103.1665,B 11.8453,C -0.0179,E1 11.8094,E2 347.4722} C_DIS
LIN {X -34.4436,Y 133.8385,Z 164,A 104.8164,B 11.8453,C -0.0193,E1 11.8049,E2 345.8102} C_DIS
LIN {X -38.5604,Y 132.7104,Z 164,A 106.5643,B 11.8453,C -0.0173,E1 11.8002,E2 344.0662} C_DIS
LIN {X -45.954,Y 130.3366,Z 164,A 109.7351,B 11.8453,C -0.0129,E1 11.7919,E2 340.9041} C_DIS
LIN {X -49.2833,Y 129.1151,Z 164,A 111.1898,B 11.8453,C -0.0109,E1 11.788,E2 339.4525} C_DIS
LIN {X -54.2832,Y 127.0927,Z 164,A 113.5295,B 11.8453,C -0.0108,E1 11.782,E2 337.1019} C_DIS
LIN {X -57.7531,Y 125.5527,Z 164,A 115.0147,B 11.8453,C -0.0066,E1 11.7782,E2 335.629} C_DIS
LIN {X -60.7636,Y 124.1241,Z 164,A 116.3911,B 11.8453,C -0.0047,E1 11.7748,E2 334.2545} C_DIS
LIN {X -63.5367,Y 122.7285,Z 164,A 117.7508,B 11.8453,C -0.0046,E1 11.7714,E2 332.887} C_DIS
LIN {X -67.453,Y 120.6216,Z 164,A 119.6533,B 11.8453,C -0.0033,E1 11.7667,E2 330.9789} C_DIS
LIN {X -71.1729,Y 118.465,Z 164,A 121.978,B 11.8453,C -0.0135,E1 11.761,E2 328.5883} C_DIS
LIN {X -75.4335,Y 115.7981,Z 164,A 124.1401,B 11.8453,C -0.012,E1 11.7559,E2 326.4183} C_DIS
LIN {X -79.8974,Y 112.7646,Z 164,A 125.7847,B 11.8453,C 0.0061,E1 11.7523,E2 324.8501} C_DIS
LIN {X -85.5602,Y 108.5306,Z 164,A 128.7368,B 11.8453,C 0.0111,E1 11.7458,E2 321.8985} C_DIS
LIN {X -88.9731,Y 105.7507,Z 164,A 130.5541,B 11.8453,C 0.0148,E1 11.7418,E2 320.084} C_DIS
LIN {X -92.2914,Y 102.8673,Z 164,A 132.8561,B 11.8453,C 0.0071,E1 11.7369,E2 317.7242} C_DIS
LIN {X -95.5574,Y 99.8407,Z 164,A 134.2738,B 11.8453,C 0.021,E1 11.7342,E2 316.362} C_DIS
LIN {X -99.5909,Y 95.8186,Z 164,A 136.7093,B 11.8453,C 0.0244,E1 11.7294,E2 313.9198} C_DIS
LIN {X -104.3358,Y 90.6284,Z 164,A 139.538,B 11.8453,C 0.033,E1 11.7241,E2 311.1052} C_DIS
LIN {X -108.0087,Y 86.218,Z 164,A 142.0553,B 11.8453,C 0.0353,E1 11.7196,E2 308.5736} C_DIS
LIN {X -110.6262,Y 82.8333,Z 164,A 143.8461,B 11.8453,C 0.0392,E1 11.7166,E2 306.7827} C_DIS
LIN {X -113.1568,Y 79.3414,Z 164,A 145.6211,B 11.8453,C 0.0438,E1 11.7137,E2 305.0113} C_DIS
LIN {X -115.6175,Y 75.7106,Z 164,A 147.4356,B 11.8453,C 0.0485,E1 11.7109,E2 303.1994} C_DIS
LIN {X -117.9611,Y 72.0046,Z 164,A 149.3147,B 11.8453,C 0.0517,E1 11.7082,E2 301.3147} C_DIS
LIN {X -120.2028,Y 68.1965,Z 164,A 151.1566,B 11.8453,C 0.0562,E1 11.7056,E2 299.4738} C_DIS
LIN {X -122.2323,Y 64.4837,Z 164,A 152.853,B 11.8452,C 0.0622,E1 11.7034,E2 297.7866} C_DIS
LIN {X -123.7572,Y 61.5073,Z 164,A 154.3158,B 11.8452,C 0.0641,E1 11.7015,E2 296.3159} C_DIS
LIN {X -125.3707,Y 58.1468,Z 164,A 155.861,B 11.8452,C 0.0683,E1 11.6997,E2 294.7725} C_DIS
LIN {X -126.8239,Y 54.9048,Z 164,A 157.2619,B 11.8452,C 0.074,E1 11.6981,E2 293.3824} C_DIS
LIN {X -127.9888,Y 52.134,Z 164,A 159.1117,B 11.8452,C 0.0636,E1 11.6961,E2 291.4584} C_DIS
LIN {X -129.7025,Y 47.7156,Z 164,A 160.5503,B 11.8451,C 0.0812,E1 11.6948,E2 290.0882} C_DIS
LIN {X -131.5466,Y 42.3613,Z 164,A 163.0297,B 11.8451,C 0.0848,E1 11.6925,E2 287.595} C_DIS
LIN {X -132.7618,Y 38.3849,Z 164,A 164.6681,B 11.845,C 0.0916,E1 11.6912,E2 285.9694} C_DIS
LIN {X -133.7739,Y 34.6983,Z 164,A 166.3632,B 11.845,C 0.0937,E1 11.69,E2 284.2624} C_DIS
LIN {X -134.6702,Y 31.0309,Z 164,A 167.9082,B 11.845,C 0.0987,E1 11.689,E2 282.7217} C_DIS
LIN {X -135.3504,Y 27.916,Z 164,A 169.1147,B 11.8449,C 0.1051,E1 11.6883,E2 281.5311} C_DIS
LIN {X -136.0159,Y 24.4666,Z 164,A 170.6656,B 11.8449,C 0.1073,E1 11.6875,E2 279.97} C_DIS
LIN {X -136.5076,Y 21.5587,Z 164,A 171.9507,B 11.8449,C 0.1094,E1 11.687,E2 278.6785} C_DIS
LIN {X -136.9899,Y 18.2422,Z 164,A 173.3762,B 11.8449,C 0.1127,E1 11.6864,E2 277.2501} C_DIS
LIN {X -137.4087,Y 14.758,Z 164,A 174.7333,B 11.8448,C 0.1192,E1 11.686,E2 275.9068} C_DIS
LIN {X -137.7055,Y 11.6685,Z 164,A 176.1516,B 11.8448,C 0.12,E1 11.6856,E2 274.4735} C_DIS
LIN {X -138.0513,Y 6.4107,Z 164,A 178.4187,B 11.8447,C 0.1246,E1 11.6853,E2 272.1985} C_DIS
LIN {X -138.1785,Y 2.3867,Z 164,A -179.7515,B 11.8447,C 0.1259,E1 11.6851,E2 270.3503} C_DIS
LIN {X -138.1648,Y -3.1522,Z 164,A -177.6394,B 11.8446,C 0.1368,E1 11.6852,E2 268.2639} C_DIS
LIN {X -138.0236,Y -6.9607,Z 164,A -176.0133,B 11.8446,C 0.1404,E1 11.6854,E2 266.6336} C_DIS
LIN {X -137.7441,Y -11.2117,Z 164,A -174.2407,B 11.8445,C 0.1455,E1 11.6858,E2 264.8621} C_DIS
LIN {X -137.4195,Y -14.658,Z 164,A -172.8126,B 11.8445,C 0.1498,E1 11.6862,E2 263.4363} C_DIS
LIN {X -136.9594,Y -18.4752,Z 164,A -171.0676,B 11.8444,C 0.151,E1 11.6868,E2 261.6739} C_DIS
LIN {X -136.3826,Y -22.3356,Z 164,A -169.535,B 11.8444,C 0.1577,E1 11.6875,E2 260.1537} C_DIS
LIN {X -135.7585,Y -25.8564,Z 164,A -168.0832,B 11.8442,C 0.1627,E1 11.6882,E2 258.7072} C_DIS
LIN {X -135.0679,Y -29.25,Z 164,A -166.5579,B 11.8442,C 0.1647,E1 11.6891,E2 257.1721} C_DIS
LIN {X -134.1233,Y -33.3213,Z 164,A -164.922,B 11.8442,C 0.1719,E1 11.6901,E2 255.55} C_DIS
LIN {X -132.0657,Y -40.7137,Z 164,A -161.5961,B 11.844,C 0.1775,E1 11.6927,E2 252.2089} C_DIS
LIN {X -130.8349,Y -44.5167,Z 164,A -159.9437,B 11.844,C 0.1822,E1 11.6941,E2 250.5586} C_DIS
LIN {X -129.1163,Y -49.2795,Z 164,A -157.7168,B 11.844,C 0.185,E1 11.6963,E2 248.3174} C_DIS
LIN {X -127.6163,Y -53.0376,Z 164,A -156.1372,B 11.8438,C 0.1918,E1 11.698,E2 246.7514} C_DIS
LIN {X -126.2623,Y -56.1849,Z 164,A -154.5281,B 11.8438,C 0.1912,E1 11.6998,E2 245.1197} C_DIS
LIN {X -124.1726,Y -60.6653,Z 164,A -152.5625,B 11.8438,C 0.1985,E1 11.7022,E2 243.1662} C_DIS
LIN {X -122.6088,Y -63.7667,Z 164,A -151.1467,B 11.8436,C 0.2028,E1 11.704,E2 241.7546} C_DIS
LIN {X -120.6562,Y -67.3914,Z 164,A -149.3425,B 11.8436,C 0.2049,E1 11.7064,E2 239.9394} C_DIS
LIN {X -118.428,Y -71.2341,Z 164,A -147.4567,B 11.8436,C 0.2084,E1 11.7091,E2 238.0492} C_DIS
LIN {X -116.3468,Y -74.5842,Z 164,A -145.407,B 11.8436,C 0.2026,E1 11.7123,E2 235.9478} C_DIS
LIN {X -113.8214,Y -78.3844,Z 164,A -143.9504,B 11.8434,C 0.2174,E1 11.7145,E2 234.5478} C_DIS
LIN {X -111.3642,Y -81.8376,Z 164,A -141.9978,B 11.8434,C 0.2168,E1 11.7177,E2 232.5714} C_DIS
LIN {X -108.0037,Y -86.2242,Z 164,A -139.8474,B 11.8432,C 0.2253,E1 11.7214,E2 230.4402} C_DIS
LIN {X -105.6961,Y -89.0381,Z 164,A -138.2665,B 11.8432,C 0.2269,E1 11.7242,E2 228.8509} C_DIS
LIN {X -101.3412,Y -93.965,Z 164,A -135.5744,B 11.8431,C 0.2335,E1 11.7292,E2 226.1646} C_DIS
LIN {X -98.325,Y -97.1171,Z 164,A -133.7025,B 11.8431,C 0.2357,E1 11.7329,E2 224.2853} C_DIS
LIN {X -95.1068,Y -100.2707,Z 164,A -131.8623,B 11.8429,C 0.24,E1 11.7366,E2 222.4495} C_DIS
LIN {X -92.0624,Y -103.0724,Z 164,A -129.5138,B 11.8432,C 0.2278,E1 11.7416,E2 220.0204} C_DIS
LIN {X -87.848,Y -106.6876,Z 164,A -127.808,B 11.8428,C 0.2465,E1 11.7451,E2 218.3919} C_DIS
LIN {X -84.3137,Y -109.5024,Z 164,A -126.0684,B 11.8427,C 0.253,E1 11.7489,E2 216.6699} C_DIS
LIN {X -81.0144,Y -111.9645,Z 164,A -124.1968,B 11.8427,C 0.2518,E1 11.7532,E2 214.7777} C_DIS
LIN {X -77.1731,Y -114.6465,Z 164,A -122.2741,B 11.8427,C 0.2553,E1 11.7576,E2 212.858} C_DIS
LIN {X -73.6321,Y -116.9518,Z 164,A -120.4845,B 11.8426,C 0.257,E1 11.7618,E2 211.0639} C_DIS
LIN {X -69.881,Y -119.2311,Z 164,A -118.6817,B 11.8426,C 0.2599,E1 11.7661,E2 209.2635} C_DIS
LIN {X -66.1605,Y -121.335,Z 164,A -116.8654,B 11.8426,C 0.2612,E1 11.7706,E2 207.4417} C_DIS
LIN {X -63.2492,Y -122.8769,Z 164,A -115.5484,B 11.8424,C 0.2641,E1 11.7738,E2 206.131} C_DIS
LIN {X -59.8502,Y -124.5667,Z 164,A -114.2114,B 11.8423,C 0.2718,E1 11.7771,E2 204.8244} C_DIS
LIN {X -55.4192,Y -126.6015,Z 164,A -111.9254,B 11.8423,C 0.2675,E1 11.783,E2 202.5047} C_DIS
LIN {X -52.3887,Y -127.8862,Z 164,A -110.5768,B 11.8423,C 0.2692,E1 11.7865,E2 201.158} C_DIS
LIN {X -49.0549,Y -129.2008,Z 164,A -108.9914,B 11.8423,C 0.2681,E1 11.7906,E2 199.5598} C_DIS
LIN {X -45.1049,Y -130.6309,Z 164,A -107.3484,B 11.8423,C 0.2721,E1 11.7949,E2 197.9292} C_DIS
LIN {X -41.0107,Y -131.9748,Z 164,A -105.6046,B 11.8423,C 0.2746,E1 11.7996,E2 196.1907} C_DIS
LIN {X -37.8496,Y -132.9162,Z 164,A -104.2053,B 11.8423,C 0.2747,E1 11.8033,E2 194.7872} C_DIS
LIN {X -34.2068,Y -133.8986,Z 164,A -102.7247,B 11.8421,C 0.2778,E1 11.8073,E2 193.317} C_DIS
LIN {X -31.0101,Y -134.6749,Z 164,A -101.3502,B 11.8421,C 0.2783,E1 11.811,E2 191.9408} C_DIS
LIN {X -27.436,Y -135.4481,Z 164,A -98.7838,B 11.8427,C 0.2517,E1 11.8184,E2 189.2381} C_DIS
LIN {X -20.5389,Y -136.6655,Z 164,A -96.7918,B 11.8422,C 0.2766,E1 11.8236,E2 187.3635} C_DIS
LIN {X -13.901,Y -137.4998,Z 164,A -93.8527,B 11.8422,C 0.2728,E1 11.8318,E2 184.4023} C_DIS
LIN {X -9.2915,Y -137.8885,Z 164,A -92.1038,B 11.8422,C 0.2774,E1 11.8366,E2 182.6744} C_DIS
LIN {X -5.8229,Y -138.077,Z 164,A -90.7105,B 11.8422,C 0.2787,E1 11.8405,E2 181.2865} C_DIS
LIN {X -0.7264,Y -138.1972,Z 164,A -88.3298,B 11.8422,C 0.2714,E1 11.8472,E2 178.8703} C_DIS
LIN {X -0.7264,Y -138.1972,Z 164,A -88.3298,B 11.8422,C 0.2714,E1 11.8472,E2 178.8703} C_DIS
Enddeposition()
LIN {X 0.9912,Y -139.1121,Z 164,A -88.2273,B 11.842,C 0.2946,E1 11.8475,E2 178.8808} C_DIS
Startdeposition()
$VEL.CP = VEL_PRINT
LIN {X -2.0978,Y -139.1031,Z 164,A -89.7772,B 11.8418,C 0.3021,E1 11.843,E2 180.4671} C_DIS
LIN {X -6.3334,Y -138.976,Z 164,A -91.4189,B 11.8418,C 0.2994,E1 11.8385,E2 182.0965} C_DIS
LIN {X -8.9016,Y -138.834,Z 164,A -92.4961,B 11.8418,C 0.2999,E1 11.8355,E2 183.1763} C_DIS
LIN {X -11.5328,Y -138.6399,Z 164,A -93.5573,B 11.8418,C 0.2991,E1 11.8325,E2 184.2347} C_DIS
LIN {X -14.265,Y -138.3867,Z 164,A -94.6855,B 11.8418,C 0.2989,E1 11.8294,E2 185.3631} C_DIS
LIN {X -18.2595,Y -137.9152,Z 164,A -96.3934,B 11.8418,C 0.2998,E1 11.8246,E2 187.0781} C_DIS
LIN {X -21.6567,Y -137.423,Z 164,A -97.8755,B 11.8418,C 0.3012,E1 11.8205,E2 188.5694} C_DIS
LIN {X -24.8373,Y -136.8838,Z 164,A -99.1957,B 11.8418,C 0.3004,E1 11.8169,E2 189.8889} C_DIS
LIN {X -30.7944,Y -135.6675,Z 164,A -101.6935,B 11.8418,C 0.2991,E1 11.8101,E2 192.3865} C_DIS
LIN {X -34.2794,Y -134.829,Z 164,A -103.4097,B 11.8418,C 0.3043,E1 11.8053,E2 194.1337} C_DIS
LIN {X -38.802,Y -133.5979,Z 164,A -105.2476,B 11.8418,C 0.3007,E1 11.8004,E2 195.9602} C_DIS
LIN {X -42.9078,Y -132.3374,Z 164,A -106.8683,B 11.842,C 0.2956,E1 11.7962,E2 197.5622} C_DIS
LIN {X -45.8875,Y -131.3329,Z 164,A -108.2517,B 11.842,C 0.2968,E1 11.7925,E2 198.9569} C_DIS
LIN {X -50.1312,Y -129.7722,Z 164,A -109.9108,B 11.8421,C 0.29,E1 11.7882,E2 200.5903} C_DIS
LIN {X -52.5603,Y -128.8086,Z 164,A -111.0982,B 11.8421,C 0.2917,E1 11.7851,E2 201.7919} C_DIS
LIN {X -55.618,Y -127.5175,Z 164,A -112.5282,B 11.8421,C 0.2918,E1 11.7814,E2 203.2299} C_DIS
LIN {X -60.2495,Y -125.3952,Z 164,A -114.623,B 11.8421,C 0.2894,E1 11.7761,E2 205.3243} C_DIS
LIN {X -63.9967,Y -123.5268,Z 164,A -116.4688,B 11.8421,C 0.2903,E1 11.7715,E2 207.1855} C_DIS
LIN {X -67.9665,Y -121.3879,Z 164,A -118.2753,B 11.8421,C 0.2866,E1 11.7671,E2 208.9853} C_DIS
LIN {X -71.6047,Y -119.2785,Z 164,A -120.0405,B 11.8422,C 0.285,E1 11.7628,E2 210.7546} C_DIS
LIN {X -75.2157,Y -117.0345,Z 164,A -121.7926,B 11.8422,C 0.2825,E1 11.7587,E2 212.5065} C_DIS
LIN {X -78.9902,Y -114.521,Z 164,A -123.6994,B 11.8423,C 0.2806,E1 11.7542,E2 214.4179} C_DIS
LIN {X -82.3135,Y -112.1557,Z 164,A -125.3953,B 11.8423,C 0.2782,E1 11.7504,E2 216.1153} C_DIS
LIN {X -86.0578,Y -109.3091,Z 164,A -127.3054,B 11.8425,C 0.2743,E1 11.7462,E2 218.0215} C_DIS
LIN {X -89.2767,Y -106.6964,Z 164,A -128.9909,B 11.8425,C 0.2707,E1 11.7426,E2 219.7037} C_DIS
LIN {X -92.7379,Y -103.702,Z 164,A -130.8098,B 11.8427,C 0.2656,E1 11.7388,E2 221.5135} C_DIS
LIN {X -95.6133,Y -101.0571,Z 164,A -132.5877,B 11.8427,C 0.2666,E1 11.7351,E2 223.3123} C_DIS
LIN {X -98.9302,Y -97.8128,Z 164,A -134.463,B 11.8427,C 0.2619,E1 11.7314,E2 225.1822} C_DIS
LIN {X -101.9234,Y -94.6892,Z 164,A -137.1452,B 11.8424,C 0.2794,E1 11.7261,E2 227.9766} C_DIS
LIN {X -106.4275,Y -89.5971,Z 164,A -138.8777,B 11.843,C 0.2483,E1 11.7232,E2 229.5737} C_DIS
LIN {X -108.5042,Y -87.071,Z 164,A -140.4947,B 11.843,C 0.2517,E1 11.7203,E2 231.2243} C_DIS
LIN {X -111.2991,Y -83.469,Z 164,A -142.1318,B 11.8432,C 0.2418,E1 11.7175,E2 232.8298} C_DIS
LIN {X -113.1329,Y -80.9652,Z 164,A -143.6705,B 11.8432,C 0.2449,E1 11.7149,E2 234.4007} C_DIS
LIN {X -115.7844,Y -77.1259,Z 164,A -145.7242,B 11.8432,C 0.2435,E1 11.7117,E2 236.4698} C_DIS
LIN {X -117.7785,Y -74.0453,Z 164,A -147.1395,B 11.8432,C 0.2376,E1 11.7096,E2 237.872} C_DIS
LIN {X -120.1581,Y -70.1186,Z 164,A -149.0808,B 11.8433,C 0.234,E1 11.7068,E2 239.8185} C_DIS
LIN {X -122.2962,Y -66.3188,Z 164,A -150.9299,B 11.8433,C 0.2307,E1 11.7043,E2 241.673} C_DIS
LIN {X -124.1865,Y -62.7039,Z 164,A -152.504,B 11.8435,C 0.224,E1 11.7023,E2 243.2324} C_DIS
LIN {X -125.6758,Y -59.662,Z 164,A -153.9231,B 11.8435,C 0.2209,E1 11.7006,E2 244.6535} C_DIS
LIN {X -127.093,Y -56.5799,Z 164,A -155.3185,B 11.8436,C 0.2171,E1 11.699,E2 246.0475} C_DIS
LIN {X -128.559,Y -53.1667,Z 164,A -156.8527,B 11.8437,C 0.2131,E1 11.6973,E2 247.5811} C_DIS
LIN {X -130.1458,Y -49.154,Z 164,A -158.4692,B 11.8439,C 0.2046,E1 11.6957,E2 249.1759} C_DIS
LIN {X -130.9549,Y -46.955,Z 164,A -159.679,B 11.8439,C 0.2076,E1 11.6945,E2 250.4157} C_DIS
LIN {X -132.0715,Y -43.716,Z 164,A -161.1043,B 11.8439,C 0.204,E1 11.6933,E2 251.8415} C_DIS
LIN {X -133.1102,Y -40.4433,Z 164,A -162.5802,B 11.8439,C 0.2015,E1 11.692,E2 253.3239} C_DIS
LIN {X -134.6367,Y -35.0364,Z 164,A -164.8144,B 11.8441,C 0.1932,E1 11.6904,E2 255.5461} C_DIS
LIN {X -135.3979,Y -31.9651,Z 164,A -166.1016,B 11.8441,C 0.1891,E1 11.6896,E2 256.83} C_DIS
LIN {X -136.0317,Y -29.1437,Z 164,A -167.3007,B 11.8441,C 0.1859,E1 11.6888,E2 258.029} C_DIS
LIN {X -136.7179,Y -25.7356,Z 164,A -168.7875,B 11.8442,C 0.183,E1 11.688,E2 259.5214} C_DIS
LIN {X -137.3334,Y -22.225,Z 164,A -170.3853,B 11.8442,C 0.1817,E1 11.6873,E2 261.134} C_DIS
LIN {X -137.8831,Y -18.5043,Z 164,A -171.7744,B 11.8443,C 0.1736,E1 11.6868,E2 262.5015} C_DIS
LIN {X -138.2606,Y -15.4366,Z 164,A -173.0558,B 11.8444,C 0.1701,E1 11.6863,E2 263.7827} C_DIS
LIN {X -138.6176,Y -11.7966,Z 164,A -174.6623,B 11.8444,C 0.1679,E1 11.6859,E2 265.4002} C_DIS
LIN {X -138.8838,Y -8.0929,Z 164,A -176.1989,B 11.8444,C 0.1636,E1 11.6856,E2 266.9361} C_DIS
LIN {X -139.0346,Y -4.8668,Z 164,A -177.5618,B 11.8445,C 0.1604,E1 11.6855,E2 268.3017} C_DIS
LIN {X -139.1126,Y 1.4088,Z 164,A 179.884,B 11.8446,C 0.1521,E1 11.6855,E2 270.8494} C_DIS
LIN {X -139.0506,Y 4.383,Z 164,A 178.4373,B 11.8446,C 0.1535,E1 11.6855,E2 272.3223} C_DIS
LIN {X -138.8274,Y 9.0096,Z 164,A 176.5938,B 11.8447,C 0.1464,E1 11.6858,E2 274.1557} C_DIS
LIN {X -138.2963,Y 15.1054,Z 164,A 174.27,B 11.8449,C 0.1346,E1 11.6864,E2 276.4523} C_DIS
LIN {X -137.9483,Y 18.0068,Z 164,A 172.8749,B 11.8449,C 0.1353,E1 11.6869,E2 277.8699} C_DIS
LIN {X -137.4158,Y 21.7033,Z 164,A 171.183,B 11.8449,C 0.1343,E1 11.6876,E2 279.5793} C_DIS
LIN {X -136.7297,Y 25.6736,Z 164,A 169.7118,B 11.8449,C 0.1252,E1 11.6883,E2 281.0251} C_DIS
LIN {X -136.1474,Y 28.6081,Z 164,A 168.4165,B 11.8449,C 0.1231,E1 11.689,E2 282.327} C_DIS
LIN {X -135.5208,Y 31.4364,Z 164,A 167.1878,B 11.845,C 0.1204,E1 11.6898,E2 283.5587} C_DIS
LIN {X -134.8058,Y 34.3707,Z 164,A 165.8518,B 11.845,C 0.1189,E1 11.6907,E2 284.9046} C_DIS
LIN {X -133.8604,Y 37.8879,Z 164,A 164.248,B 11.845,C 0.1169,E1 11.6919,E2 286.5196} C_DIS
LIN {X -132.7819,Y 41.5159,Z 164,A 162.8234,B 11.8451,C 0.1095,E1 11.6931,E2 287.9259} C_DIS
LIN {X -131.9906,Y 43.9588,Z 164,A 161.6632,B 11.8451,C 0.1088,E1 11.6941,E2 289.0974} C_DIS
LIN {X -130.7081,Y 47.6393,Z 164,A 159.9731,B 11.8451,C 0.1062,E1 11.6957,E2 290.7962} C_DIS
LIN {X -128.6827,Y 52.8705,Z 164,A 157.8037,B 11.8452,C 0.0966,E1 11.6979,E2 292.9456} C_DIS
LIN {X -126.9231,Y 56.9599,Z 164,A 155.8896,B 11.8452,C 0.0934,E1 11.7,E2 294.8673} C_DIS
LIN {X -125.2628,Y 60.5266,Z 164,A 154.2928,B 11.8452,C 0.0885,E1 11.702,E2 296.4594} C_DIS
LIN {X -123.7157,Y 63.6288,Z 164,A 152.849,B 11.8453,C 0.0851,E1 11.7038,E2 297.9036} C_DIS
LIN {X -122.0948,Y 66.6879,Z 164,A 151.3465,B 11.8453,C 0.0831,E1 11.7058,E2 299.4139} C_DIS
LIN {X -120.1249,Y 70.175,Z 164,A 149.6142,B 11.8453,C 0.0807,E1 11.7082,E2 301.1546} C_DIS
LIN {X -117.7796,Y 74.0434,Z 164,A 147.7449,B 11.8453,C 0.0761,E1 11.7109,E2 303.0225} C_DIS
LIN {X -115.2746,Y 77.8858,Z 164,A 145.8446,B 11.8453,C 0.0716,E1 11.7139,E2 304.922} C_DIS
LIN {X -112.636,Y 81.655,Z 164,A 143.8138,B 11.8453,C 0.0701,E1 11.7172,E2 306.9674} C_DIS
LIN {X -109.1081,Y 86.3128,Z 164,A 141.175,B 11.8454,C 0.0697,E1 11.7218,E2 309.6321} C_DIS
LIN {X -106.6087,Y 89.3811,Z 164,A 139.7845,B 11.8454,C 0.0604,E1 11.7242,E2 310.9913} C_DIS
LIN {X -102.6242,Y 93.9296,Z 164,A 137.4682,B 11.8454,C 0.0508,E1 11.7284,E2 313.2834} C_DIS
LIN {X -100.1372,Y 96.5765,Z 164,A 135.8254,B 11.8454,C 0.0509,E1 11.7316,E2 314.9427} C_DIS
LIN {X -97.08,Y 99.6498,Z 164,A 133.9213,B 11.8454,C 0.0499,E1 11.7354,E2 316.8595} C_DIS
Enddeposition()
END
